idx:=1;
MessageHandler.MessageLine[idx].Visible:=FALSE;
MessageHandler.MessageLine[idx].Editable:=TRUE;
MessageHandler.MessageLine[idx].Text:='Specialmode_1';				(*Ablauf Pallettierer*)
MessageHandler.MessageLine[idx].MsgInt:=1;
MessageHandler.MessageLine[idx].MsgBool:=FALSE;
MessageHandler.MessageLine[idx].MsgTypeEnum:=MsgDataTypeBool;

idx:=idx+1;
MessageHandler.MessageLine[idx].Visible:=FALSE;
MessageHandler.MessageLine[idx].Editable:=TRUE;
MessageHandler.MessageLine[idx].Text:='Specialmode_2';				(*Not used*)
MessageHandler.MessageLine[idx].MsgInt:=2;
MessageHandler.MessageLine[idx].MsgBool:=FALSE;
MessageHandler.MessageLine[idx].MsgTypeEnum:=MsgDataTypeBool;

idx:=idx+1;
MessageHandler.MessageLine[idx].Visible:=FALSE;
MessageHandler.MessageLine[idx].Editable:=TRUE;
MessageHandler.MessageLine[idx].Text:='Specialmode_3';				(*Not used*)
MessageHandler.MessageLine[idx].MsgInt:=3;
MessageHandler.MessageLine[idx].MsgBool:=FALSE;
MessageHandler.MessageLine[idx].MsgTypeEnum:=MsgDataTypeBool;

idx:=idx+1;
MessageHandler.MessageLine[idx].Visible:=FALSE;
MessageHandler.MessageLine[idx].Editable:=TRUE;
MessageHandler.MessageLine[idx].Text:='Specialmode_4';				(*Not used*)
MessageHandler.MessageLine[idx].MsgInt:=4;
MessageHandler.MessageLine[idx].MsgBool:=FALSE;
MessageHandler.MessageLine[idx].MsgTypeEnum:=MsgDataTypeBool;

idx:=idx+1;
MessageHandler.MessageLine[idx].Visible:=FALSE;
MessageHandler.MessageLine[idx].Editable:=TRUE;
MessageHandler.MessageLine[idx].Text:='Specialmode_5';				(*Blister Abstapeln*)
MessageHandler.MessageLine[idx].MsgInt:=5;
MessageHandler.MessageLine[idx].MsgBool:=FALSE;
MessageHandler.MessageLine[idx].MsgTypeEnum:=MsgDataTypeBool;

idx:=idx+1;
MessageHandler.MessageLine[idx].Visible:=gTypeCode=312 OR gTypeCode=499 OR gTypeCode=322;	(*93pol*)(*102pol*)(*160pol*);
MessageHandler.MessageLine[idx].Editable:=TRUE;
MessageHandler.MessageLine[idx].Text:='Specialmode_6';				(*Dummytest*)
MessageHandler.MessageLine[idx].MsgInt:=6;
MessageHandler.MessageLine[idx].MsgBool:=FALSE;
MessageHandler.MessageLine[idx].MsgTypeEnum:=MsgDataTypeBool;

idx:=idx+1;
MessageHandler.MessageLine[idx].Visible:=FALSE;
MessageHandler.MessageLine[idx].Editable:=TRUE;
MessageHandler.MessageLine[idx].Text:='Specialmode_7';				(*Not used*)
MessageHandler.MessageLine[idx].MsgInt:=7;
MessageHandler.MessageLine[idx].MsgBool:=FALSE;
MessageHandler.MessageLine[idx].MsgTypeEnum:=MsgDataTypeBool;

idx:=idx+1;
MessageHandler.MessageLine[idx].Visible:=FALSE;
MessageHandler.MessageLine[idx].Editable:=TRUE;
MessageHandler.MessageLine[idx].Text:='Specialmode_8';				(*Not used*)
MessageHandler.MessageLine[idx].MsgInt:=8;
MessageHandler.MessageLine[idx].MsgBool:=FALSE;
MessageHandler.MessageLine[idx].MsgTypeEnum:=MsgDataTypeBool;

IF 	ModeNo>=1 AND
	ModeNo<=8 THEN
	MessageHandler.MessageLine[ModeNo].MsgBool:=TRUE;
END_IF
END_ACTION

ACTION Msg_SpecialMenu_action:
MessageHandler.Msg.ID:='PM61';
MessageHandler.Msg.Name:='Teil-Abläufe';
MessageHandler.Msg.Text:='Teilablauf auswählen und mit OK starten';
MessageHandler.Msg.Color:=Color.yellow;
MessageHandler.Msg.Station:=0;


MessageHandler(
	Prio:=2, 					(*1=highest, .. , 4=lowest*)
	Btn1Addr:=ADR(MsgOk),		(*Address of Button1 , if Zero then Button is unvisible*)
	Btn2Addr:=ADR(MsgCancel),	(*Address of Button2 , if Zero then Button is unvisible*)
	sVisu:=Visu.Message);

MessageHandler.DisableMultiSelect(sVisu:=Visu.Message);

FOR idx:=1 TO 10 DO
	IF 	MessageHandler.MessageLine[idx].MsgBool THEN
		ModeNo:=idx;
	END_IF
END_FOR
END_ACTION

ACTION Msg_SpecialMenu_exit:
MsgOk:=FALSE;
MsgCancel:=FALSE;
END_ACTION

ACTION SpecialMode01__action:
IF SpecialMode01.State=STATE_WAIT
THEN
	SpecialMode01(Start:=TRUE);

	SFCRun:=TRUE;
(*ELSE*)
END_IF
END_ACTION

ACTION SpecialMode01__exit:
SpecialMode01.Start:=FALSE;
SFCRun:=FALSE;
END_ACTION

ACTION SpecialMode02__action:
IF SpecialMode02.State=STATE_WAIT
THEN
	SpecialMode02(Start:=TRUE);

	SFCRun:=TRUE;
(*ELSE*)
END_IF
END_ACTION

ACTION SpecialMode02__exit:
SpecialMode02.Start:=FALSE;
SFCRun:=FALSE;
END_ACTION

ACTION SpecialMode03__action:
IF SpecialMode03.State=STATE_WAIT
THEN
	SpecialMode03(Start:=TRUE);

	SFCRun:=TRUE;
(*ELSE*)
END_IF
END_ACTION

ACTION SpecialMode03__exit:
SpecialMode03.Start:=FALSE;
SFCRun:=FALSE;
END_ACTION

ACTION SpecialMode04__action:
IF SpecialMode04.State=STATE_WAIT
THEN
	SpecialMode04(Start:=TRUE);

	SFCRun:=TRUE;
(*ELSE*)
END_IF
END_ACTION

ACTION SpecialMode04__exit:
SpecialMode04.Start:=FALSE;
SFCRun:=FALSE;
END_ACTION

ACTION SpecialMode05__action:
IF SpecialMode05.State=STATE_WAIT
THEN
	SpecialMode05(Start:=TRUE);

	SFCRun:=TRUE;
(*ELSE*)
END_IF
END_ACTION

ACTION SpecialMode05__exit:
SpecialMode05.Start:=FALSE;
SFCRun:=FALSE;
END_ACTION

ACTION SpecialMode06__action:
IF SpecialMode06.State=STATE_WAIT
THEN
	SpecialMode06(Start:=TRUE);

	IF	gTypeCode=312 OR		(*93pol*)
		gTypeCode=499 THEN		(*102pol*)
		MP.ST02.DummyPruefung_93pol  := TRUE;
	ELSIF
		gTypeCode=322	THEN	(*160pol*)
		DummyTest_160pol := TRUE;
	END_IF
	SFCRun:=TRUE;
END_IF
END_ACTION

ACTION SpecialMode06__exit:
SpecialMode06.Start:=FALSE;
SFCRun:=FALSE;
DummyTest_160pol := FALSE;
MP.ST02.DummyPruefung_93pol  := FALSE;
END_ACTION

ACTION SpecialMode07__action:
IF SpecialMode07.State=STATE_WAIT
THEN
	SpecialMode07(Start:=TRUE);

	SFCRun:=TRUE;
(*ELSE*)
END_IF
END_ACTION

ACTION SpecialMode07__exit:
SpecialMode07.Start:=FALSE;
SFCRun:=FALSE;
END_ACTION

ACTION SpecialMode08__action:
IF SpecialMode08.State=STATE_WAIT
THEN
	SpecialMode08(Start:=TRUE);

	SFCRun:=TRUE;
(*ELSE*)
END_IF
END_ACTION

ACTION SpecialMode08__exit:
SpecialMode08.Start:=FALSE;
SFCRun:=FALSE;
END_ACTION

ACTION SeqEnd_action:
SFCTime:=TIME_TO_DINT(TIME()-SFCTimeStart);
State:=STATE_OK;
END_ACTION

TRANSITION ModeNo=1:
ModeNo=1
END_TRANSITION

TRANSITION StateOk:
		SFCRun=TRUE
AND SpecialMode01.State=STATE_OK
END_TRANSITION

TRANSITION ModeNo=2:
ModeNo=2
END_TRANSITION

TRANSITION StateOk:
		SFCRun=TRUE
AND SpecialMode02.State=STATE_OK
END_TRANSITION

TRANSITION ModeNo=3:
ModeNo=3
END_TRANSITION

TRANSITION StateOk:
		SFCRun=TRUE
AND SpecialMode03.State=STATE_OK
END_TRANSITION

TRANSITION ModeNo=4:
ModeNo=4
END_TRANSITION

TRANSITION StateOk:
		SFCRun=TRUE
AND SpecialMode04.State=STATE_OK
END_TRANSITION

TRANSITION ModeNo=5:
ModeNo=5
END_TRANSITION

TRANSITION StateOk:
		SFCRun=TRUE
AND SpecialMode05.State=STATE_OK
END_TRANSITION

TRANSITION ModeNo=6:
ModeNo=6
END_TRANSITION

TRANSITION StateOk:
		SFCRun=TRUE
AND SpecialMode06.State=STATE_OK
END_TRANSITION

TRANSITION ModeNo=7:
ModeNo=7
END_TRANSITION

TRANSITION StateOk:
		SFCRun=TRUE
AND SpecialMode07.State=STATE_OK
END_TRANSITION

TRANSITION ModeNo=8:
ModeNo=8
END_TRANSITION

TRANSITION StateOk:
		SFCRun=TRUE
AND SpecialMode08.State=STATE_OK
END_TRANSITION
END_PROGRAM

(* POU Stations/ST_00/ST00_SFCs/_SpecialModeSFCs/SpecialMode02, SFC *)
PROGRAM SpecialMode02 (*Used for: Prozess Kamera *)
(* Date:     Author:   *)

VAR_OUTPUT
	SFCCurrentPOU		: STRING:='SpecialMode02';
	SFCCurrentStep	: STRING:='';
	SFCTime					:	DINT;
  State   				:	DINT;
  Result  				:	DINT;
END_VAR
VAR_INPUT
	Start						:	BOOL;
END_VAR
VAR
	MsgOK				:	BOOL;
	MsgCancel		:	BOOL;
	SFCRun					:	BOOL;
	SFCTimeStart		:	TIME;

	(* Userdefinded area *)


END_VAR
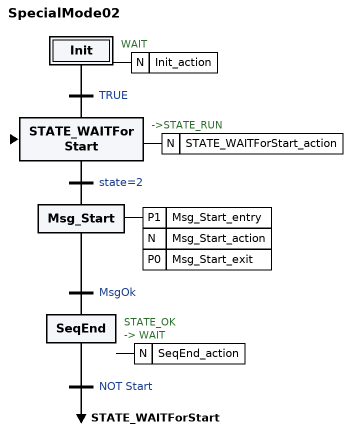
INITIAL_STEP Init: (* WAIT *)
	Init_action(N);
END_STEP
TRANSITION FROM Init TO STATE_WAITForStart := TRUE;
END_TRANSITION
STEP STATE_WAITForStart: (* ->STATE_RUN *)
	STATE_WAITForStart_action(N);
END_STEP
TRANSITION FROM STATE_WAITForStart TO Msg_Start := state=2;
END_TRANSITION
STEP Msg_Start:
	Msg_Start_entry(P1);
	Msg_Start_action(N);
	Msg_Start_exit(P0);
END_STEP
TRANSITION FROM Msg_Start TO SeqEnd := MsgOk;
END_TRANSITION
STEP SeqEnd: (* STATE_OK / -> WAIT *)
	SeqEnd_action(N);
END_STEP
TRANSITION FROM SeqEnd TO STATE_WAITForStart := NOT Start;
END_TRANSITION

ACTION Init_action:
Start:=FALSE;
State:=STATE_WAIT;
END_ACTION

ACTION STATE_WAITForStart_action:
IF Start=TRUE
THEN
	State:=STATE_RUN;
	Result:=RESULT_NON;
	SFCTimeStart:=TIME();
(*ELSE*)
END_IF
END_ACTION

ACTION Msg_Start_entry:
MessageHandler.ClearMessageLines(sVisu:=Visu.Message);
END_ACTION

ACTION Msg_Start_action:
MessageHandler.Msg.ID:='PM51';
MessageHandler.Msg.Name:='SpecialMode02_Start';
MessageHandler.Msg.Text:='Special Mode 2';
MessageHandler.Msg.Color:=Color.yellow;
MessageHandler.Msg.Station:=1;


MessageHandler(
	Prio:=2, 									(*1=highest, .. , 4=lowest*)
	Btn1Addr:=ADR(MsgOk),			(*Address of Button1 , if Zero then Button is unvisible*)
	Btn2Addr:=ADR(MsgCancel),	(*Address of Button2 , if Zero then Button is unvisible*)
	sVisu:=Visu.Message);


MessageHandler.MessageLine[1].Visible:=TRUE;
MessageHandler.MessageLine[1].Editable:=TRUE;
MessageHandler.MessageLine[1].Text:='Kamera Programm ';
MessageHandler.MessageLine[1].MsgTypeEnum:=MsgDataTypeDint;
END_ACTION

ACTION Msg_Start_exit:
MsgOk:=FALSE;
MsgCancel:=FALSE;
SpecialModeProgNu:=MessageHandler.MessageLine[1].MsgInt;
END_ACTION

ACTION SeqEnd_action:
IF 	State=STATE_RUN THEN
	SFCTime:=TIME_TO_DINT(TIME()-SFCTimeStart);
	State:=STATE_OK;
END_IF

IF 	NOT Start THEN
	State:=STATE_WAIT;
END_IF
END_ACTION
END_PROGRAM

(* POU Stations/ST_00/ST00_SFCs/_SpecialModeSFCs/SpecialMode04, SFC *)
PROGRAM SpecialMode04 (*not used*)
(* Date:     Author:   *)

VAR_OUTPUT
	SFCCurrentPOU		: STRING:='SpecialMode04';
	SFCCurrentStep		: STRING:='';
	SFCTime				: DINT;
	State   			: DINT;
	Result  			: DINT;
END_VAR
VAR_INPUT
	Start				: BOOL;
END_VAR
VAR
	MsgOK				: BOOL;
	MsgCancel			: BOOL;
	SFCRun				: BOOL;
	SFCTimeStart		: TIME;
	ResultString		: STRING;
	(* Userdefinded area *)



END_VAR
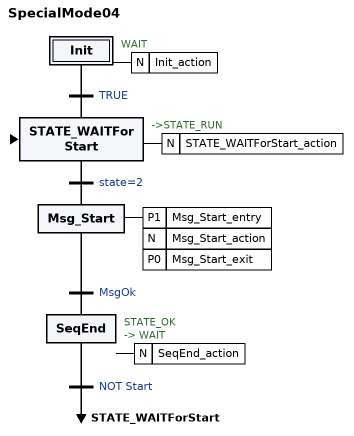
INITIAL_STEP Init: (* WAIT *)
	Init_action(N);
END_STEP
TRANSITION FROM Init TO STATE_WAITForStart := TRUE;
END_TRANSITION
STEP STATE_WAITForStart: (* ->STATE_RUN *)
	STATE_WAITForStart_action(N);
END_STEP
TRANSITION FROM STATE_WAITForStart TO Msg_Start := state=2;
END_TRANSITION
STEP Msg_Start:
	Msg_Start_entry(P1);
	Msg_Start_action(N);
	Msg_Start_exit(P0);
END_STEP
TRANSITION FROM Msg_Start TO SeqEnd := MsgOk;
END_TRANSITION
STEP SeqEnd: (* STATE_OK / -> WAIT *)
	SeqEnd_action(N);
END_STEP
TRANSITION FROM SeqEnd TO STATE_WAITForStart := NOT Start;
END_TRANSITION

ACTION Init_action:
Start:=FALSE;
State:=STATE_WAIT;
END_ACTION

ACTION STATE_WAITForStart_action:
IF Start=TRUE
THEN
	State:=STATE_RUN;
	Result:=RESULT_NON;
	SFCTimeStart:=TIME();
(*ELSE*)
END_IF
END_ACTION

ACTION Msg_Start_entry:
MessageHandler.ClearMessageLines(sVisu:=Visu.Message);
END_ACTION

ACTION Msg_Start_action:
MessageHandler.Msg.ID:='PM52';
MessageHandler.Msg.Name:='SpecialMode04_Start';
MessageHandler.Msg.Text:='Special Mode 4';
MessageHandler.Msg.Color:=Color.yellow;
MessageHandler.Msg.Station:=1;


MessageHandler(
	Prio:=2, 									(*1=highest, .. , 4=lowest*)
	Btn1Addr:=ADR(MsgOk),			(*Address of Button1 , if Zero then Button is unvisible*)
	Btn2Addr:=ADR(MsgCancel),	(*Address of Button2 , if Zero then Button is unvisible*)
	sVisu:=Visu.Message);


MessageHandler.MessageLine[1].Visible:=TRUE;
MessageHandler.MessageLine[1].Editable:=TRUE;
MessageHandler.MessageLine[1].Text:='Kamera Programm ';
MessageHandler.MessageLine[1].MsgTypeEnum:=MsgDataTypeDint;
END_ACTION

ACTION Msg_Start_exit:
MsgOk:=FALSE;
MsgCancel:=FALSE;

SpecialModeProgNu:=MessageHandler.MessageLine[1].MsgInt;
END_ACTION

ACTION SeqEnd_action:
IF 	State=STATE_RUN THEN
	SFCTime:=TIME_TO_DINT(TIME()-SFCTimeStart);
	State:=STATE_OK;
END_IF

IF 	NOT Start THEN
	State:=STATE_WAIT;
END_IF
END_ACTION
END_PROGRAM

(* POU Stations/ST_00/ST00_SFCs/_SpecialModeSFCs/SpecialMode05, SFC *)
PROGRAM SpecialMode05 (*Used for: xxxx *)
(* Date:     Author:   *)

VAR_OUTPUT
	SFCCurrentPOU		: STRING:='SpecialMode05';
	SFCCurrentStep	: STRING:='';
	SFCTime					:	DINT;
  State   				:	DINT;
  Result  				:	DINT;

	ConveyorOn				: BOOL;

END_VAR
VAR_INPUT
	Start						:	BOOL;
END_VAR
VAR
	MsgOK				:	BOOL;
	MsgCancel		:	BOOL;
	SFCRun					:	BOOL;
	SFCTimeStart		:	TIME;

	(* Userdefinded area *)

END_VAR
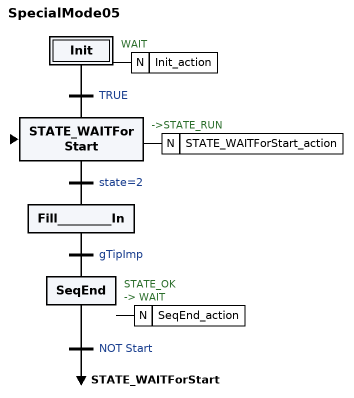
INITIAL_STEP Init: (* WAIT *)
	Init_action(N);
END_STEP
TRANSITION FROM Init TO STATE_WAITForStart := TRUE;
END_TRANSITION
STEP STATE_WAITForStart: (* ->STATE_RUN *)
	STATE_WAITForStart_action(N);
END_STEP
TRANSITION FROM STATE_WAITForStart TO Fill_________In := state=2;
END_TRANSITION
STEP Fill_________In:
END_STEP
TRANSITION FROM Fill_________In TO SeqEnd := gTipImp;
END_TRANSITION
STEP SeqEnd: (* STATE_OK / -> WAIT *)
	SeqEnd_action(N);
END_STEP
TRANSITION FROM SeqEnd TO STATE_WAITForStart := NOT Start;
END_TRANSITION

ACTION Init_action:
Start:=FALSE;
State:=STATE_WAIT;
END_ACTION

ACTION STATE_WAITForStart_action:
IF Start=TRUE
THEN
	State:=STATE_RUN;
	Result:=RESULT_NON;
	SFCTimeStart:=TIME();
(*ELSE*)
END_IF
END_ACTION

ACTION SeqEnd_action:
IF 	State=STATE_RUN THEN
	SFCTime:=TIME_TO_DINT(TIME()-SFCTimeStart);
	State:=STATE_OK;
END_IF

IF 	NOT Start THEN
	State:=STATE_WAIT;
END_IF
END_ACTION
END_PROGRAM

(* POU Stations/ST_00/ST00_SFCs/_SpecialModeSFCs/SpecialMode07, SFC *)
PROGRAM SpecialMode07 (*Used for: xxxx *)
(* Date:     Author:   *)

VAR_OUTPUT
	SFCCurrentPOU		: STRING:='SpecialMode07';
	SFCCurrentStep	: STRING:='';
	SFCTime					:	DINT;
  State   				:	DINT;
  Result  				:	DINT;
END_VAR
VAR_INPUT
	Start						:	BOOL;
END_VAR
VAR
	MsgOK				:	BOOL;
	MsgCancel		:	BOOL;
	SFCRun					:	BOOL;
	SFCTimeStart		:	TIME;
  Delay         :TON;

	(* Userdefinded area *)


END_VAR
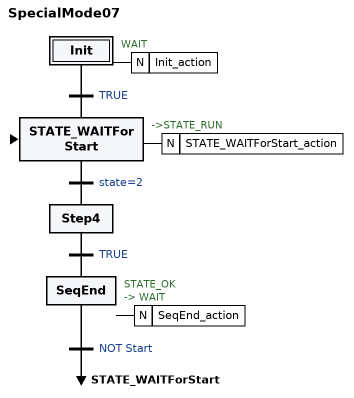
INITIAL_STEP Init: (* WAIT *)
	Init_action(N);
END_STEP
TRANSITION FROM Init TO STATE_WAITForStart := TRUE;
END_TRANSITION
STEP STATE_WAITForStart: (* ->STATE_RUN *)
	STATE_WAITForStart_action(N);
END_STEP
TRANSITION FROM STATE_WAITForStart TO Step4 := state=2;
END_TRANSITION
STEP Step4:
END_STEP
TRANSITION FROM Step4 TO SeqEnd := TRUE;
END_TRANSITION
STEP SeqEnd: (* STATE_OK / -> WAIT *)
	SeqEnd_action(N);
END_STEP
TRANSITION FROM SeqEnd TO STATE_WAITForStart := NOT Start;
END_TRANSITION

ACTION Init_action:
Start:=FALSE;
State:=STATE_WAIT;
END_ACTION

ACTION STATE_WAITForStart_action:
IF Start=TRUE
THEN
	State:=STATE_RUN;
	Result:=RESULT_NON;
	SFCTimeStart:=TIME();
(*ELSE*)
END_IF
END_ACTION

ACTION SeqEnd_action:
IF 	State=STATE_RUN THEN
	SFCTime:=TIME_TO_DINT(TIME()-SFCTimeStart);
	State:=STATE_OK;
END_IF

IF 	NOT Start THEN
	State:=STATE_WAIT;
END_IF
END_ACTION
END_PROGRAM

(* POU Stations/ST_00/ST00_SFCs/_SpecialModeSFCs/SpecialMode08, SFC *)
PROGRAM SpecialMode08 (*Used for: xxxx *)
(* Date:     Author:   *)

VAR_OUTPUT
	SFCCurrentPOU		: STRING:='SpecialMode08';
	SFCCurrentStep	: STRING:='';
	SFCTime					:	DINT;
  State   				:	DINT;
  Result  				:	DINT;
END_VAR
VAR_INPUT
	Start						:	BOOL;
END_VAR
VAR
	MsgOK				:	BOOL;
	MsgCancel		:	BOOL;
	SFCRun					:	BOOL;
	SFCTimeStart		:	TIME;

	(* Userdefinded area *)
	TestDint1:DINT:=12;
	TestDint2:DINT:=34;
	IntPosIdx:	DINT;

END_VAR
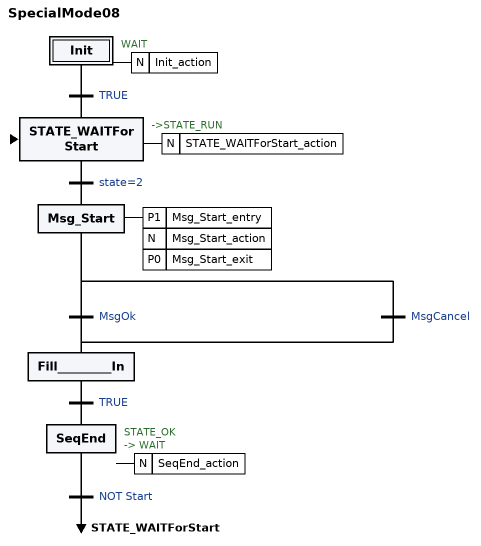
INITIAL_STEP Init: (* WAIT *)
	Init_action(N);
END_STEP
TRANSITION FROM Init TO STATE_WAITForStart := TRUE;
END_TRANSITION
STEP STATE_WAITForStart: (* ->STATE_RUN *)
	STATE_WAITForStart_action(N);
END_STEP
TRANSITION FROM STATE_WAITForStart TO Msg_Start := state=2;
END_TRANSITION
STEP Msg_Start:
	Msg_Start_entry(P1);
	Msg_Start_action(N);
	Msg_Start_exit(P0);
END_STEP
TRANSITION FROM Msg_Start TO Fill_________In := MsgOk;
END_TRANSITION
TRANSITION FROM Msg_Start TO Fill_________In := MsgCancel;
END_TRANSITION
STEP Fill_________In:
END_STEP
TRANSITION FROM Fill_________In TO SeqEnd := TRUE;
END_TRANSITION
STEP SeqEnd: (* STATE_OK / -> WAIT *)
	SeqEnd_action(N);
END_STEP
TRANSITION FROM SeqEnd TO STATE_WAITForStart := NOT Start;
END_TRANSITION

ACTION Init_action:
Start:=FALSE;
State:=STATE_WAIT;
END_ACTION

ACTION STATE_WAITForStart_action:
IF Start=TRUE
THEN
	State:=STATE_RUN;
	Result:=RESULT_NON;
	SFCTimeStart:=TIME();
(*ELSE*)
END_IF
END_ACTION

ACTION Msg_Start_entry:
MessageHandler.ClearMessageLines(sVisu:=Visu.Message);
IntPosIdx:=1;
END_ACTION

ACTION Msg_Start_action:
MessageHandler.Msg.ID:='PM53';
MessageHandler.Msg.Name:='SpecialMode08_Start';
MessageHandler.Msg.Text:='Teilautomatik Ablauf08: Test Messagehandler';
MessageHandler.Msg.Color:=Color.yellow;
MessageHandler.Msg.Station:=1;


MessageHandler(
	Prio:=2, 									(*1=highest, .. , 4=lowest*)
	Btn1Addr:=ADR(MsgOk),			(*Address of Button1 , if Zero then Button is unvisible*)
	Btn2Addr:=ADR(MsgCancel),	(*Address of Button2 , if Zero then Button is unvisible*)
	sVisu:=Visu.Message);


MessageHandler.MessageLine[1].Visible:=TRUE;
MessageHandler.MessageLine[1].Editable:=TRUE;
MessageHandler.MessageLine[1].Text:='TestZeile1';
MessageHandler.MessageLine[1].MsgInt:=TestDint1;
MessageHandler.MessageLine[1].MsgTypeEnum:=MsgDataTypeDint;

MessageHandler.MessageLine[2].Visible:=TRUE;
MessageHandler.MessageLine[2].Editable:=TRUE;
MessageHandler.MessageLine[2].Text:='TestZeile2';
MessageHandler.MessageLine[2].MsgInt:=TestDint2;
MessageHandler.MessageLine[2].MsgTypeEnum:=MsgDataTypeDint;
END_ACTION

ACTION Msg_Start_exit:
MsgOk:=FALSE;
MsgCancel:=FALSE;

TestDint1:=MessageHandler.MessageLine[1].MsgInt;
TestDint2:=MessageHandler.MessageLine[2].MsgInt;
END_ACTION

ACTION SeqEnd_action:
IF 	State=STATE_RUN THEN
	SFCTime:=TIME_TO_DINT(TIME()-SFCTimeStart);
	State:=STATE_OK;
END_IF


IF 	NOT Start THEN
	State:=STATE_WAIT;
END_IF
END_ACTION
END_PROGRAM

(* POU Stations/ST_00/ST00_SFCs/HomePositionSFC, SFC *)
PROGRAM HomePositionSFC


VAR_OUTPUT
	SFCCurrentPOU		: STRING:='HomePositionSFC';
	SFCCurrentStep		: STRING:='';
	SFCTime				: DINT;
	State   			: StateObject	:= STATE_WAIT;
	Result  			: StateResult;
END_VAR
VAR_INPUT
	Start				: BOOL;
END_VAR
VAR
	MsgOK				: BOOL;
	MsgCancel			: BOOL;
	SFCRun				: BOOL;
	SFCTimeStart		: TIME;
	Error				: ErrorStruct;
	(* Userdefinded area *)
	SFCRun01			: BOOL;
	SFCRun02			: BOOL;
	SFCRun03			: BOOL;
	SFCRun04			: BOOL;
	SFCRun05			: BOOL;
	SFCRun08			: BOOL;
	idx					: INT;


END_VAR
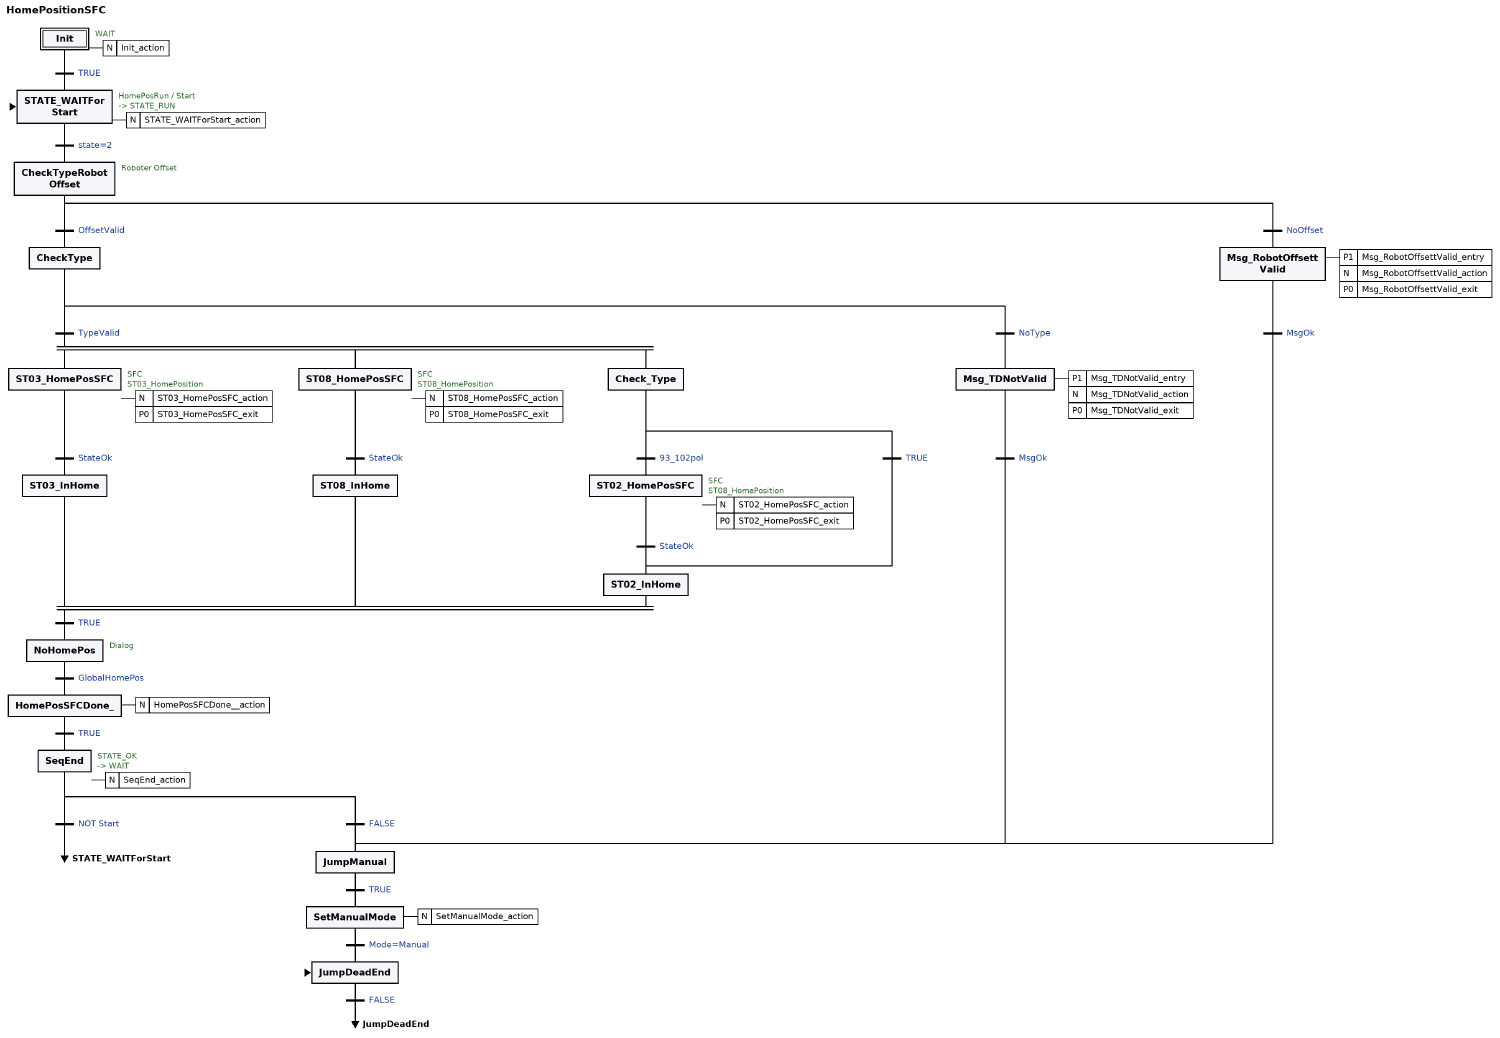
INITIAL_STEP Init: (* WAIT *)
	Init_action(N);
END_STEP
TRANSITION FROM Init TO STATE_WAITForStart := TRUE;
END_TRANSITION
STEP STATE_WAITForStart: (* HomePosRun / Start / -> STATE_RUN *)
	STATE_WAITForStart_action(N);
END_STEP
TRANSITION FROM STATE_WAITForStart TO CheckTypeRobotOffset := state=2;
END_TRANSITION
STEP CheckTypeRobotOffset: (* Roboter Offset *)
END_STEP
TRANSITION FROM CheckTypeRobotOffset TO CheckType := OffsetValid;
END_TRANSITION
TRANSITION FROM CheckTypeRobotOffset TO Msg_RobotOffsettValid := NoOffset;
END_TRANSITION
STEP CheckType:
END_STEP
TRANSITION FROM CheckType TO (ST03_HomePosSFC, ST08_HomePosSFC, Check_Type) := TypeValid;
END_TRANSITION
TRANSITION FROM CheckType TO Msg_TDNotValid := NoType;
END_TRANSITION
STEP Msg_TDNotValid:
	Msg_TDNotValid_entry(P1);
	Msg_TDNotValid_action(N);
	Msg_TDNotValid_exit(P0);
END_STEP
TRANSITION FROM Msg_TDNotValid TO JumpManual := MsgOk;
END_TRANSITION
STEP Msg_RobotOffsettValid:
	Msg_RobotOffsettValid_entry(P1);
	Msg_RobotOffsettValid_action(N);
	Msg_RobotOffsettValid_exit(P0);
END_STEP
TRANSITION FROM Msg_RobotOffsettValid TO JumpManual := MsgOk;
END_TRANSITION
STEP ST03_HomePosSFC: (* SFC / ST03_HomePosition *)
	ST03_HomePosSFC_action(N);
	ST03_HomePosSFC_exit(P0);
END_STEP
TRANSITION FROM ST03_HomePosSFC TO ST03_InHome := StateOk;
END_TRANSITION
STEP ST03_InHome:
END_STEP
STEP ST08_HomePosSFC: (* SFC / ST08_HomePosition *)
	ST08_HomePosSFC_action(N);
	ST08_HomePosSFC_exit(P0);
END_STEP
TRANSITION FROM ST08_HomePosSFC TO ST08_InHome := StateOk;
END_TRANSITION
STEP ST08_InHome:
END_STEP
STEP Check_Type:
END_STEP
TRANSITION FROM Check_Type TO ST02_HomePosSFC := 93_102pol;
END_TRANSITION
TRANSITION FROM Check_Type TO ST02_InHome := TRUE;
END_TRANSITION
STEP ST02_HomePosSFC: (* SFC / ST08_HomePosition *)
	ST02_HomePosSFC_action(N);
	ST02_HomePosSFC_exit(P0);
END_STEP
TRANSITION FROM ST02_HomePosSFC TO ST02_InHome := StateOk;
END_TRANSITION
STEP ST02_InHome:
END_STEP
TRANSITION FROM (ST03_InHome, ST08_InHome, ST02_InHome) TO NoHomePos := TRUE;
END_TRANSITION
STEP NoHomePos: (* Dialog *)
END_STEP
TRANSITION FROM NoHomePos TO HomePosSFCDone_ := GlobalHomePos;
END_TRANSITION
STEP HomePosSFCDone_:
	HomePosSFCDone__action(N);
END_STEP
TRANSITION FROM HomePosSFCDone_ TO SeqEnd := TRUE;
END_TRANSITION
STEP SeqEnd: (* STATE_OK / -> WAIT *)
	SeqEnd_action(N);
END_STEP
TRANSITION FROM SeqEnd TO STATE_WAITForStart := NOT Start;
END_TRANSITION
TRANSITION FROM SeqEnd TO JumpManual := FALSE;
END_TRANSITION
STEP JumpManual:
END_STEP
TRANSITION FROM JumpManual TO SetManualMode := TRUE;
END_TRANSITION
STEP SetManualMode:
	SetManualMode_action(N);
END_STEP
TRANSITION FROM SetManualMode TO JumpDeadEnd := Mode=Manual;
END_TRANSITION
STEP JumpDeadEnd:
END_STEP
TRANSITION FROM JumpDeadEnd TO JumpDeadEnd := FALSE;
END_TRANSITION

ACTION Init_action:
Start:=FALSE;
State:=STATE_WAIT;
END_ACTION

ACTION STATE_WAITForStart_action:
IF	(ModeSelect.Mode=MODE_HOME_POS_RUN OR
	Start) AND
	NOT PLC_PRG.GlobalHomePos THEN
	State:=STATE_RUN;
	Result:=RESULT_NON;
	SFCTimeStart:=TIME();
END_IF

SFCRun		:=FALSE;
SFCRun01	:=FALSE;
SFCRun02	:=FALSE;
SFCRun03	:=FALSE;
SFCRun04	:=FALSE;
SFCRun05	:=FALSE;
END_ACTION

ACTION Msg_TDNotValid_entry:
FOR idx:=1 TO 8
DO
	MessageHandler.MessageLine[idx].Visible:=FALSE;
	MessageHandler.MessageLine[idx].Editable:=FALSE;
	MessageHandler.MessageLine[idx].Text:='';
	MessageHandler.MessageLine[idx].MsgInt:=0;
	MessageHandler.MessageLine[idx].MsgTypeEnum:=MsgDataTypeDint;

END_FOR
END_ACTION

ACTION Msg_TDNotValid_action:
MessageHandler.Msg.ID:='PM10';
MessageHandler.Msg.Name:='TDNotValid';
MessageHandler.Msg.Text:='Typdaten nicht gültig, bitte laden!';
MessageHandler.Msg.Text:= CONCAT(MessageHandler.Msg.Text,'$r --> weiter mit <OK>');
MessageHandler.Msg.Color:=Color.yellow;
MessageHandler.Msg.Station:=0;
MessageHandler.MsgButton1Text:='continue';

MessageHandler(
	Prio:=1, 						(*1=highest, .. , 4=lowest*)
	Btn1Addr:=ADR(MsgOk),		(*Address of Button1 , if Zero then Button is unvisible*)
	Btn2Addr:=0,					(*Address of Button2 , if Zero then Button is unvisible*)
	sVisu:=Visu.Message);
END_ACTION

ACTION Msg_TDNotValid_exit:
MsgOk:=FALSE;
MsgCancel:=FALSE;
END_ACTION

ACTION Msg_RobotOffsettValid_entry:
MessageHandler.ClearMessageLines(sVisu:=Visu.Message);
END_ACTION

ACTION Msg_RobotOffsettValid_action:
MessageHandler.Msg.ID:='PM11';
MessageHandler.Msg.Name:='TDRoffsetbotOValid';
MessageHandler.Msg.Text:='Typdaten Roboter Offset nicht gültig, bitte laden!';
MessageHandler.Msg.Text:= CONCAT(MessageHandler.Msg.Text,'$r --> weiter mit <OK>');

MessageHandler.Msg.Color:=Color.yellow;
MessageHandler.Msg.Station:=0;


MessageHandler(
	Prio:=1, 								(*1=highest, .. , 4=lowest*)
	Btn1Addr:=ADR(MsgOk),		(*Address of Button1 , if Zero then Button is unvisible*)
	Btn2Addr:=0,						(*Address of Button2 , if Zero then Button is unvisible*)
	sVisu:=Visu.Message);
END_ACTION

ACTION Msg_RobotOffsettValid_exit:
MsgOk:=FALSE;
MsgCancel:=FALSE;
END_ACTION

ACTION ST03_HomePosSFC_action:
IF ST03_HomePosition.State=STATE_WAIT
THEN
	ST03_HomePosition(Start:=TRUE);

	SFCRun03:=TRUE;
(*ELSE*)
END_IF
END_ACTION

ACTION ST03_HomePosSFC_exit:
ST03_HomePosition.Start:=FALSE;
SFCRun03:=FALSE;
END_ACTION

ACTION ST08_HomePosSFC_action:
IF ST08_HomePosition.State=STATE_WAIT
THEN
	SFCRun08:=TRUE;
	ST08_HomePosition.Start:=TRUE;


(*ELSE*)
END_IF
END_ACTION

ACTION ST08_HomePosSFC_exit:
ST08_HomePosition.Start:=FALSE;
SFCRun08:=FALSE;
END_ACTION

ACTION ST02_HomePosSFC_action:
IF ST02_HomePosition.State=STATE_WAIT THEN
	ST02_HomePosition.Start:=TRUE;
	SFCRun02:=TRUE;
END_IF
END_ACTION

ACTION ST02_HomePosSFC_exit:
ST02_HomePosition.Start:=FALSE;
SFCRun02:=FALSE;
END_ACTION

ACTION HomePosSFCDone__action:
gHomePosSFCDone:=TRUE;
END_ACTION

ACTION SeqEnd_action:
IF 	NOT Start THEN
	State:=STATE_WAIT;
END_IF
END_ACTION

ACTION SetManualMode_action:
ModeSelect.AskForManual:=TRUE;
END_ACTION

TRANSITION OffsetValid:
   gRobotOffset > 0
(*OR gRobotOffset =1000
OR gRobotOffset =2000
OR gRobotOffset =3000
OR gRobotOffset =4000
OR gRobotOffset =5000
OR gRobotOffset =6000
OR gRobotOffset =7000
OR gRobotOffset =19000
OR gRobotOffset =25000
OR gRobotOffset =26000
OR gRobotOffset =27000
OR gRobotOffset =28000
OR gRobotOffset =29000
OR gRobotOffset =30000
OR gRobotOffset =35000*)
END_TRANSITION

TRANSITION TypeValid:
gTypeDataValid
END_TRANSITION

TRANSITION NoType:
TRUE
END_TRANSITION

TRANSITION NoOffset:
TRUE
END_TRANSITION

TRANSITION StateOk:
		SFCRun03=TRUE
AND ST03_HomePosition.State=STATE_OK
END_TRANSITION

TRANSITION StateOk:
		SFCRun08=TRUE
AND ST08_HomePosition.State=STATE_OK
END_TRANSITION

TRANSITION 93_102pol:
gTypeCode=4991 OR 	(*102pol*)
gTypeCode=312		(*93pol*)
END_TRANSITION

TRANSITION StateOk:
SFCRun02 AND
ST02_HomePosition.State=STATE_OK
END_TRANSITION

TRANSITION GlobalHomePos:
PLC_PRG.GlobalHomePos
END_TRANSITION

TRANSITION Mode=Manual:
ModeSelect.Mode=MODE_MANUAL
END_TRANSITION
END_PROGRAM

(* POU Stations/ST_03_Ruestsaetze/ST_03_SFCs/ST03_HomePosition, SFC *)
PROGRAM ST03_HomePosition

VAR_OUTPUT
	SFCCurrentPOU		: STRING:='ST03_HomePosition';
	SFCCurrentStep		: STRING:='';
	SFCTime				: DINT;
	State   			: StateObject	:= STATE_WAIT;
	Result  			: StateResult;

END_VAR
VAR_INPUT
	Start				: BOOL;
END_VAR
VAR
	MsgOK				: BOOL;
	MsgCancel			: BOOL;
	SFCRun				: BOOL;
	SFCTimeStart		: TIME;
	(* Userdefinded area *)

END_VAR
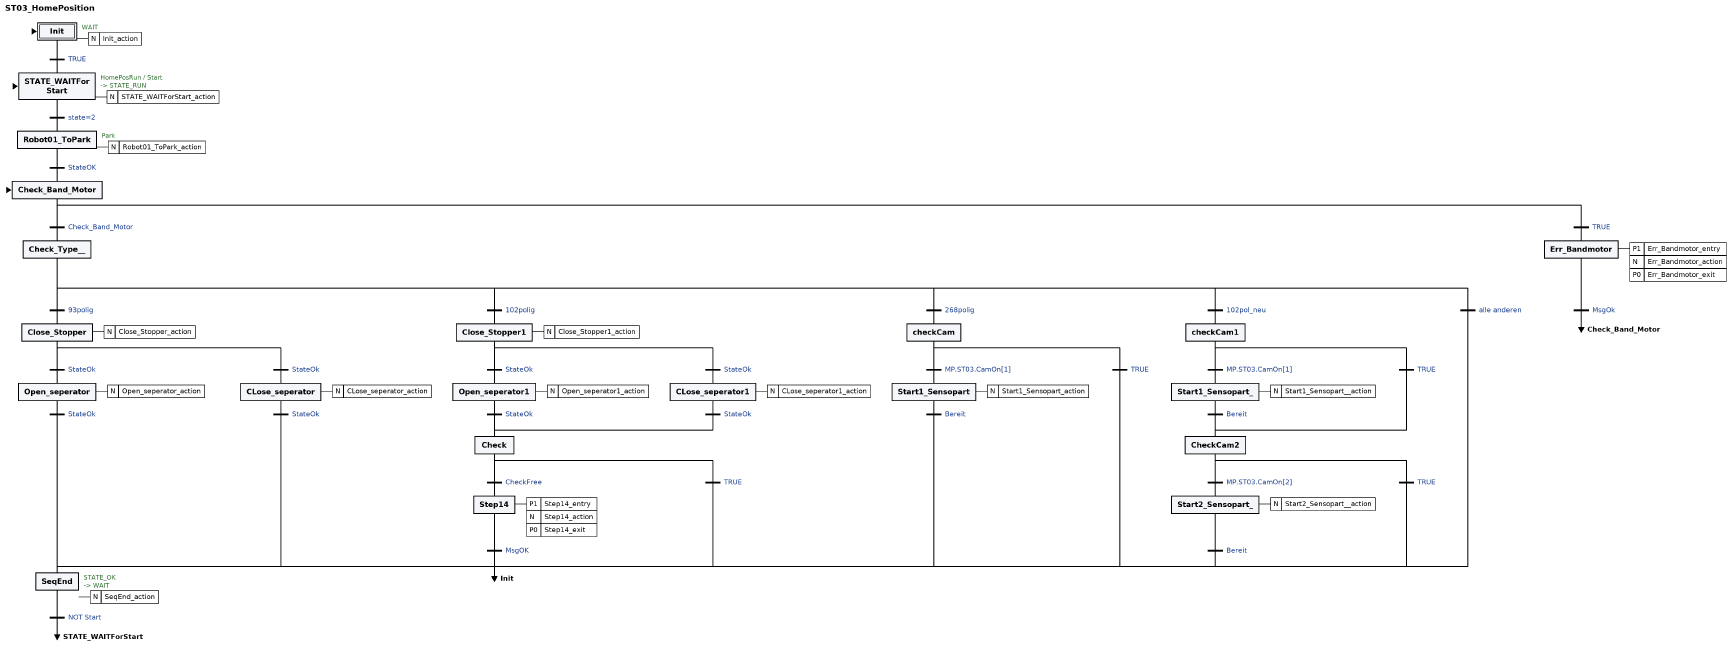
INITIAL_STEP Init: (* WAIT *)
	Init_action(N);
END_STEP
TRANSITION FROM Init TO STATE_WAITForStart := TRUE;
END_TRANSITION
STEP STATE_WAITForStart: (* HomePosRun / Start / -> STATE_RUN *)
	STATE_WAITForStart_action(N);
END_STEP
TRANSITION FROM STATE_WAITForStart TO Robot01_ToPark := state=2;
END_TRANSITION
STEP Robot01_ToPark: (* Park *)
	Robot01_ToPark_action(N);
END_STEP
TRANSITION FROM Robot01_ToPark TO Check_Band_Motor := StateOK;
END_TRANSITION
STEP Check_Band_Motor:
END_STEP
TRANSITION FROM Check_Band_Motor TO Check_Type__ := Check_Band_Motor;
END_TRANSITION
TRANSITION FROM Check_Band_Motor TO Err_Bandmotor := TRUE;
END_TRANSITION
STEP Err_Bandmotor:
	Err_Bandmotor_entry(P1);
	Err_Bandmotor_action(N);
	Err_Bandmotor_exit(P0);
END_STEP
TRANSITION FROM Err_Bandmotor TO Check_Band_Motor := MsgOk;
END_TRANSITION
STEP Check_Type__:
END_STEP
TRANSITION FROM Check_Type__ TO Close_Stopper := 93polig;
END_TRANSITION
TRANSITION FROM Check_Type__ TO Close_Stopper1 := 102polig;
END_TRANSITION
TRANSITION FROM Check_Type__ TO checkCam := 268polig;
END_TRANSITION
TRANSITION FROM Check_Type__ TO checkCam1 := 102pol_neu;
END_TRANSITION
TRANSITION FROM Check_Type__ TO SeqEnd := alle anderen;
END_TRANSITION
STEP Close_Stopper:
	Close_Stopper_action(N);
END_STEP
TRANSITION FROM Close_Stopper TO Open_seperator := StateOk;
END_TRANSITION
TRANSITION FROM Close_Stopper TO CLose_seperator := StateOk;
END_TRANSITION
STEP Open_seperator:
	Open_seperator_action(N);
END_STEP
TRANSITION FROM Open_seperator TO SeqEnd := StateOk;
END_TRANSITION
STEP CLose_seperator:
	CLose_seperator_action(N);
END_STEP
TRANSITION FROM CLose_seperator TO SeqEnd := StateOk;
END_TRANSITION
STEP Close_Stopper1:
	Close_Stopper1_action(N);
END_STEP
TRANSITION FROM Close_Stopper1 TO Open_seperator1 := StateOk;
END_TRANSITION
TRANSITION FROM Close_Stopper1 TO CLose_seperator1 := StateOk;
END_TRANSITION
STEP Open_seperator1:
	Open_seperator1_action(N);
END_STEP
TRANSITION FROM Open_seperator1 TO Check := StateOk;
END_TRANSITION
STEP CLose_seperator1:
	CLose_seperator1_action(N);
END_STEP
TRANSITION FROM CLose_seperator1 TO Check := StateOk;
END_TRANSITION
STEP Check:
END_STEP
TRANSITION FROM Check TO Step14 := CheckFree;
END_TRANSITION
TRANSITION FROM Check TO SeqEnd := TRUE;
END_TRANSITION
STEP Step14:
	Step14_entry(P1);
	Step14_action(N);
	Step14_exit(P0);
END_STEP
TRANSITION FROM Step14 TO Init := MsgOK;
END_TRANSITION
STEP checkCam:
END_STEP
TRANSITION FROM checkCam TO Start1_Sensopart := MP.ST03.CamOn[1];
END_TRANSITION
TRANSITION FROM checkCam TO SeqEnd := TRUE;
END_TRANSITION
STEP Start1_Sensopart:
	Start1_Sensopart_action(N);
END_STEP
TRANSITION FROM Start1_Sensopart TO SeqEnd := Bereit;
END_TRANSITION
STEP checkCam1:
END_STEP
TRANSITION FROM checkCam1 TO Start1_Sensopart_ := MP.ST03.CamOn[1];
END_TRANSITION
TRANSITION FROM checkCam1 TO CheckCam2 := TRUE;
END_TRANSITION
STEP Start1_Sensopart_:
	Start1_Sensopart__action(N);
END_STEP
TRANSITION FROM Start1_Sensopart_ TO CheckCam2 := Bereit;
END_TRANSITION
STEP CheckCam2:
END_STEP
TRANSITION FROM CheckCam2 TO Start2_Sensopart_ := MP.ST03.CamOn[2];
END_TRANSITION
TRANSITION FROM CheckCam2 TO SeqEnd := TRUE;
END_TRANSITION
STEP Start2_Sensopart_:
	Start2_Sensopart__action(N);
END_STEP
TRANSITION FROM Start2_Sensopart_ TO SeqEnd := Bereit;
END_TRANSITION
STEP SeqEnd: (* STATE_OK / -> WAIT *)
	SeqEnd_action(N);
END_STEP
TRANSITION FROM SeqEnd TO STATE_WAITForStart := NOT Start;
END_TRANSITION

ACTION Init_action:
Start:=FALSE;
State:=STATE_WAIT;
END_ACTION

ACTION STATE_WAITForStart_action:
IF	( Start = TRUE )
THEN
	State:=STATE_RUN;
	Result:=RESULT_NON;
	SFCTimeStart:=TIME();
ELSE
	;
END_IF
END_ACTION

ACTION Robot01_ToPark_action:
Robot01.PosNo:=POS_PARK;
Robot01.PosOffset:=gRobotOffset;
Robot01.Override:=MP.ST00.Override;
Robot01.SetToolOn:=FALSE;
Robot01.SetToolOff:=FALSE;
Robot01.ExecuteMove:=TRUE;
END_ACTION

ACTION Err_Bandmotor_entry:
MessageHandler.ClearMessageLines(sVisu:=Visu.Message);
END_ACTION

ACTION Err_Bandmotor_action:
MessageHandler.Msg.ID:='PM100';
MessageHandler.Msg.Name:='Fehler Bandmotor';
MessageHandler.Msg.Text:='Fehler Bandmotor';
MessageHandler.Msg.Color:=Color.red;
MessageHandler.Msg.Station:=1;


MessageHandler(
	Prio:=2, 							(*1=highest, .. , 4=lowest*)
	Btn1Addr:=ADR(MsgOk),			(*Address of Button1 , if Zero then Button is unvisible*)
	Btn2Addr:=,						(*Address of Button2 , if Zero then Button is unvisible*)
	sVisu:=Visu.Message);
END_ACTION

ACTION Err_Bandmotor_exit:
MsgOk:=FALSE;
MsgCancel:=FALSE;
ST03_51_M1.Reset:=TRUE;
END_ACTION

ACTION Close_Stopper_action:
ST00_74_Y2_4.MoveInit:=TRUE;
END_ACTION

ACTION Open_seperator_action:
ST00_74_Y2_5.MoveInit:=TRUE;
END_ACTION

ACTION CLose_seperator_action:
ST00_74_Y2_5.MoveWork:=TRUE;
END_ACTION

ACTION Close_Stopper1_action:
ST00_74_Y2_4.MoveInit:=TRUE;
END_ACTION

ACTION Open_seperator1_action:
ST00_74_Y2_5.MoveInit:=TRUE;
END_ACTION

ACTION CLose_seperator1_action:
ST00_74_Y2_5.MoveWork:=TRUE;
END_ACTION

ACTION Step14_entry:
MessageHandler.ClearMessageLines(sVisu:=Visu.Message);
END_ACTION

ACTION Step14_action:
MessageHandler.Msg.ID:='PM102';
MessageHandler.Msg.Name:='Vereinzler beide Positionen besetzt';
MessageHandler.Msg.Text:='Vereinzler beide Positionen besetzt';
MessageHandler.Msg.Color:=Color.red;
MessageHandler.Msg.Station:=1;


MessageHandler(
	Prio:=2, 							(*1=highest, .. , 4=lowest*)
	Btn1Addr:=ADR(MsgOk),			(*Address of Button1 , if Zero then Button is unvisible*)
	Btn2Addr:=,						(*Address of Button2 , if Zero then Button is unvisible*)
	sVisu:=Visu.Message);
END_ACTION

ACTION Step14_exit:
MsgOk:=FALSE;
MsgCancel:=FALSE;
END_ACTION

ACTION Start1_Sensopart_action:
ST03_8_100_A1.JobNo := TD.Sensopart_CamProgNo ;
ST03_8_100_A1.st_ctrl_in.b_init := TRUE;
END_ACTION

ACTION Start1_Sensopart__action:
ST03_8_100_A1.JobNo := TD.Sensopart_CamProgNo ;
ST03_8_100_A1.st_ctrl_in.b_init := TRUE;
END_ACTION

ACTION Start2_Sensopart__action:
ST03_8_103_A1.JobNo := TD.Sensopart2_CamProgNo ;
ST03_8_103_A1.st_ctrl_in.b_init := TRUE;
END_ACTION

ACTION SeqEnd_action:
IF 	State=STATE_RUN THEN
	SFCTime:=TIME_TO_DINT(TIME()-SFCTimeStart);
	State:=STATE_OK;
END_IF

IF 	NOT Start THEN
	State:=STATE_WAIT;
END_IF
END_ACTION

TRANSITION StateOK:
Robot01.State=STATE_OK
END_TRANSITION

TRANSITION Check_Band_Motor:
NOT ST03_51_M1.Error_ (*AND
ST03_51_M1.On*)
END_TRANSITION

TRANSITION 93polig:
gTypeCode=312	(*93pol*)
END_TRANSITION

TRANSITION StateOk:
ST00_74_Y2_4.State=STATE_OK AND
NOT ST00_72_X1_3.BitInToCheck
END_TRANSITION

TRANSITION StateOk:
ST00_74_Y2_5.State=STATE_OK
END_TRANSITION

TRANSITION StateOk:
ST00_74_Y2_4.State=STATE_OK
END_TRANSITION

TRANSITION StateOk:
ST00_74_Y2_5.State=STATE_OK
END_TRANSITION

TRANSITION 102polig:
gTypeCode=4991	(*102pol*)
END_TRANSITION

TRANSITION StateOk:
ST00_74_Y2_4.State=STATE_OK AND
NOT ST02_FDB_80_B02.BitInToCheck
END_TRANSITION

TRANSITION StateOk:
ST00_74_Y2_5.State=STATE_OK
END_TRANSITION

TRANSITION StateOk:
ST00_74_Y2_4.State=STATE_OK
END_TRANSITION

TRANSITION StateOk:
ST00_74_Y2_5.State=STATE_OK
END_TRANSITION

TRANSITION CheckFree:
ST02_FDB_80_B02.BitInToCheck AND
ST00_72_X1_3.BitInToCheck
END_TRANSITION

TRANSITION 268polig:
gTypeCode=5841 	(*268pol*)
END_TRANSITION

TRANSITION Bereit:
ST03_8_100_A1.st_ctrl_out.b_bereit (*Kamera Farberkennung Ehternet*)
END_TRANSITION

TRANSITION 102pol_neu:
gTypeCode=4993	(*102pol neu*)
END_TRANSITION

TRANSITION Bereit:
ST03_8_100_A1.st_ctrl_out.b_bereit  (*Kamera Farberkennung Ehternet*)
END_TRANSITION

TRANSITION Bereit:
ST03_8_103_A1.st_ctrl_out.b_bereit  (*Kamera Farberkennung Ehternet*)
END_TRANSITION

TRANSITION alle anderen:
TRUE
END_TRANSITION
END_PROGRAM

(* POU Stations/ST_08_Palettierer/ST_08_SFCs/ST08_HomePosition, SFC *)
PROGRAM ST08_HomePosition


VAR_OUTPUT
	SFCCurrentPOU		: STRING:='ST08_HomePosition';
	SFCCurrentStep		: STRING:='';
	SFCTime				: DINT;
	State   			: StateObject	:= STATE_WAIT;
	Result  			: StateResult;
END_VAR
VAR_INPUT
	Start				: BOOL;
END_VAR
VAR
	MsgOK				: BOOL;
	MsgCancel			: BOOL;
	SFCRun				: BOOL;
	SFCTimeStart		: TIME;
	(* Userdefinded area *)
	MsgString      		:STRING;
	MsgID		      	:STRING(20);
END_VAR
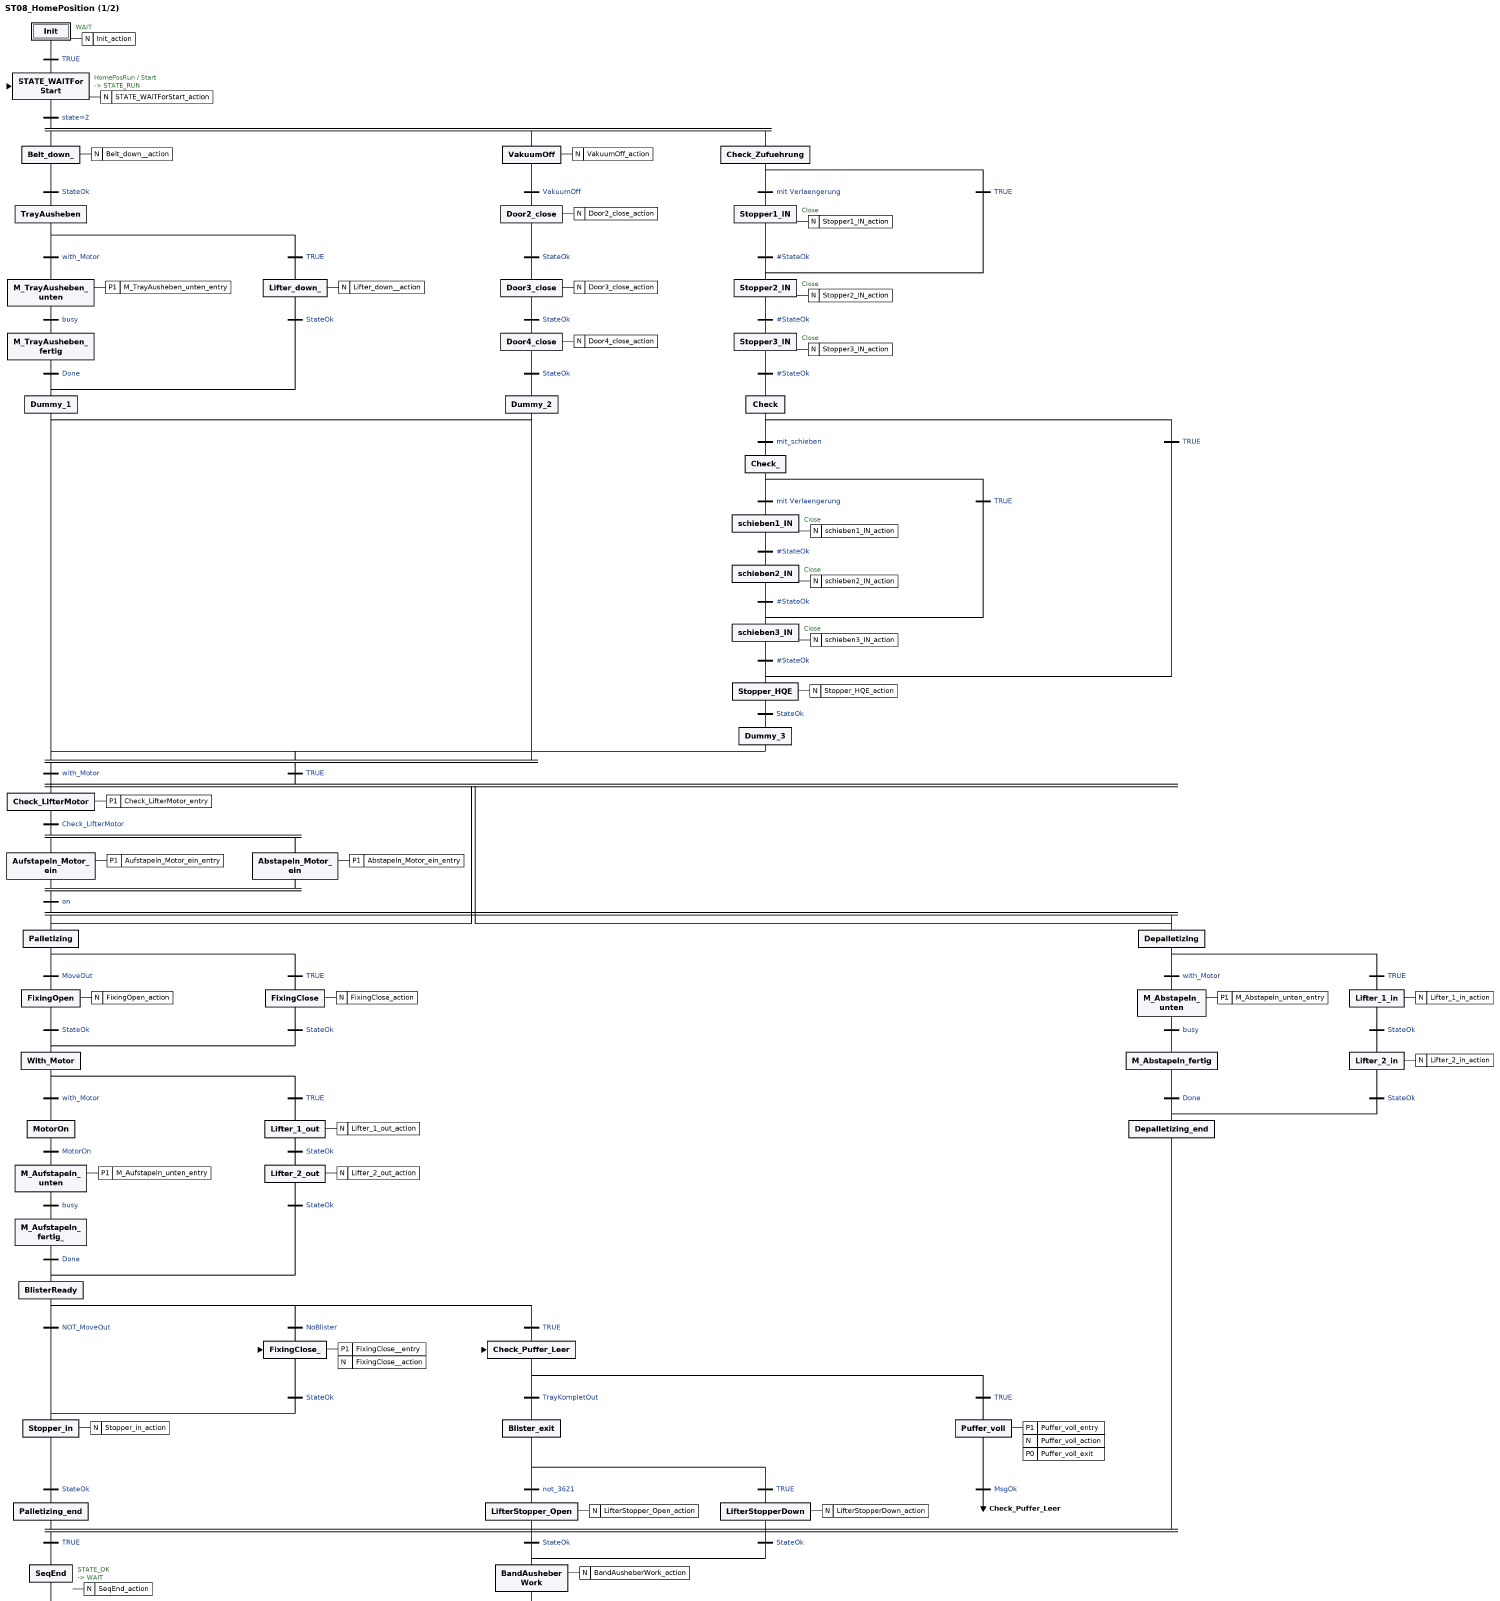
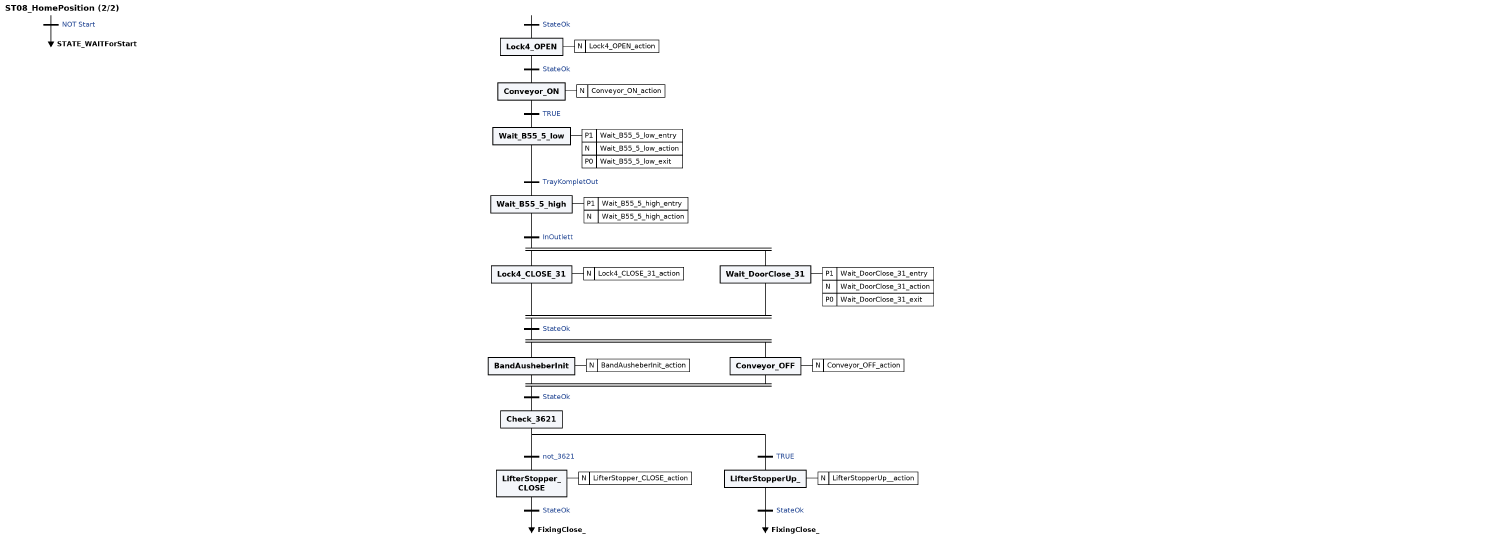
INITIAL_STEP Init: (* WAIT *)
	Init_action(N);
END_STEP
TRANSITION FROM Init TO STATE_WAITForStart := TRUE;
END_TRANSITION
STEP STATE_WAITForStart: (* HomePosRun / Start / -> STATE_RUN *)
	STATE_WAITForStart_action(N);
END_STEP
TRANSITION FROM STATE_WAITForStart TO (Belt_down_, VakuumOff, Check_Zufuehrung) := state=2;
END_TRANSITION
STEP Belt_down_:
	Belt_down__action(N);
END_STEP
TRANSITION FROM Belt_down_ TO TrayAusheben := StateOk;
END_TRANSITION
STEP TrayAusheben:
END_STEP
TRANSITION FROM TrayAusheben TO M_TrayAusheben_unten := with_Motor;
END_TRANSITION
TRANSITION FROM TrayAusheben TO Lifter_down_ := TRUE;
END_TRANSITION
STEP M_TrayAusheben_unten:
	M_TrayAusheben_unten_entry(P1);
END_STEP
TRANSITION FROM M_TrayAusheben_unten TO M_TrayAusheben_fertig := busy;
END_TRANSITION
STEP M_TrayAusheben_fertig:
END_STEP
TRANSITION FROM M_TrayAusheben_fertig TO Dummy_1 := Done;
END_TRANSITION
STEP Lifter_down_:
	Lifter_down__action(N);
END_STEP
TRANSITION FROM Lifter_down_ TO Dummy_1 := StateOk;
END_TRANSITION
STEP Dummy_1:
END_STEP
STEP VakuumOff:
	VakuumOff_action(N);
END_STEP
TRANSITION FROM VakuumOff TO Door2_close := VakuumOff;
END_TRANSITION
STEP Door2_close:
	Door2_close_action(N);
END_STEP
TRANSITION FROM Door2_close TO Door3_close := StateOk;
END_TRANSITION
STEP Door3_close:
	Door3_close_action(N);
END_STEP
TRANSITION FROM Door3_close TO Door4_close := StateOk;
END_TRANSITION
STEP Door4_close:
	Door4_close_action(N);
END_STEP
TRANSITION FROM Door4_close TO Dummy_2 := StateOk;
END_TRANSITION
STEP Dummy_2:
END_STEP
STEP Check_Zufuehrung:
END_STEP
TRANSITION FROM Check_Zufuehrung TO Stopper1_IN := mit Verlaengerung;
END_TRANSITION
TRANSITION FROM Check_Zufuehrung TO Stopper2_IN := TRUE;
END_TRANSITION
STEP Stopper1_IN: (* Close *)
	Stopper1_IN_action(N);
END_STEP
TRANSITION FROM Stopper1_IN TO Stopper2_IN := #StateOk;
END_TRANSITION
STEP Stopper2_IN: (* Close *)
	Stopper2_IN_action(N);
END_STEP
TRANSITION FROM Stopper2_IN TO Stopper3_IN := #StateOk;
END_TRANSITION
STEP Stopper3_IN: (* Close *)
	Stopper3_IN_action(N);
END_STEP
TRANSITION FROM Stopper3_IN TO Check := #StateOk;
END_TRANSITION
STEP Check:
END_STEP
TRANSITION FROM Check TO Check_ := mit_schieben;
END_TRANSITION
TRANSITION FROM Check TO Stopper_HQE := TRUE;
END_TRANSITION
STEP Check_:
END_STEP
TRANSITION FROM Check_ TO schieben1_IN := mit Verlaengerung;
END_TRANSITION
TRANSITION FROM Check_ TO schieben3_IN := TRUE;
END_TRANSITION
STEP schieben1_IN: (* Close *)
	schieben1_IN_action(N);
END_STEP
TRANSITION FROM schieben1_IN TO schieben2_IN := #StateOk;
END_TRANSITION
STEP schieben2_IN: (* Close *)
	schieben2_IN_action(N);
END_STEP
TRANSITION FROM schieben2_IN TO schieben3_IN := #StateOk;
END_TRANSITION
STEP schieben3_IN: (* Close *)
	schieben3_IN_action(N);
END_STEP
TRANSITION FROM schieben3_IN TO Stopper_HQE := #StateOk;
END_TRANSITION
STEP Stopper_HQE:
	Stopper_HQE_action(N);
END_STEP
TRANSITION FROM Stopper_HQE TO Dummy_3 := StateOk;
END_TRANSITION
STEP Dummy_3:
END_STEP
TRANSITION FROM (Dummy_1, Dummy_2, Dummy_3) TO Check_LifterMotor := with_Motor;
END_TRANSITION
TRANSITION FROM (Dummy_1, Dummy_2, Dummy_3) TO (Palletizing, Depalletizing) := TRUE;
END_TRANSITION
STEP Check_LifterMotor:
	Check_LifterMotor_entry(P1);
END_STEP
TRANSITION FROM Check_LifterMotor TO (Aufstapeln_Motor_ein, Abstapeln_Motor_ein) := Check_LifterMotor;
END_TRANSITION
STEP Aufstapeln_Motor_ein:
	Aufstapeln_Motor_ein_entry(P1);
END_STEP
STEP Abstapeln_Motor_ein:
	Abstapeln_Motor_ein_entry(P1);
END_STEP
TRANSITION FROM (Aufstapeln_Motor_ein, Abstapeln_Motor_ein) TO (Palletizing, Depalletizing) := on;
END_TRANSITION
STEP Palletizing:
END_STEP
TRANSITION FROM Palletizing TO FixingOpen := MoveOut;
END_TRANSITION
TRANSITION FROM Palletizing TO FixingClose := TRUE;
END_TRANSITION
STEP FixingOpen:
	FixingOpen_action(N);
END_STEP
TRANSITION FROM FixingOpen TO With_Motor := StateOk;
END_TRANSITION
STEP FixingClose:
	FixingClose_action(N);
END_STEP
TRANSITION FROM FixingClose TO With_Motor := StateOk;
END_TRANSITION
STEP With_Motor:
END_STEP
TRANSITION FROM With_Motor TO MotorOn := with_Motor;
END_TRANSITION
TRANSITION FROM With_Motor TO Lifter_1_out := TRUE;
END_TRANSITION
STEP MotorOn:
END_STEP
TRANSITION FROM MotorOn TO M_Aufstapeln_unten := MotorOn;
END_TRANSITION
STEP M_Aufstapeln_unten:
	M_Aufstapeln_unten_entry(P1);
END_STEP
TRANSITION FROM M_Aufstapeln_unten TO M_Aufstapeln_fertig_ := busy;
END_TRANSITION
STEP M_Aufstapeln_fertig_:
END_STEP
TRANSITION FROM M_Aufstapeln_fertig_ TO BlisterReady := Done;
END_TRANSITION
STEP Lifter_1_out:
	Lifter_1_out_action(N);
END_STEP
TRANSITION FROM Lifter_1_out TO Lifter_2_out := StateOk;
END_TRANSITION
STEP Lifter_2_out:
	Lifter_2_out_action(N);
END_STEP
TRANSITION FROM Lifter_2_out TO BlisterReady := StateOk;
END_TRANSITION
STEP BlisterReady:
END_STEP
TRANSITION FROM BlisterReady TO Stopper_in := NOT_MoveOut;
END_TRANSITION
TRANSITION FROM BlisterReady TO FixingClose_ := NoBlister;
END_TRANSITION
TRANSITION FROM BlisterReady TO Check_Puffer_Leer := TRUE;
END_TRANSITION
STEP FixingClose_:
	FixingClose__entry(P1);
	FixingClose__action(N);
END_STEP
TRANSITION FROM FixingClose_ TO Stopper_in := StateOk;
END_TRANSITION
STEP Check_Puffer_Leer:
END_STEP
TRANSITION FROM Check_Puffer_Leer TO Blister_exit := TrayKompletOut;
END_TRANSITION
TRANSITION FROM Check_Puffer_Leer TO Puffer_voll := TRUE;
END_TRANSITION
STEP Puffer_voll:
	Puffer_voll_entry(P1);
	Puffer_voll_action(N);
	Puffer_voll_exit(P0);
END_STEP
TRANSITION FROM Puffer_voll TO Check_Puffer_Leer := MsgOk;
END_TRANSITION
STEP Blister_exit:
END_STEP
TRANSITION FROM Blister_exit TO LifterStopper_Open := not_3621;
END_TRANSITION
TRANSITION FROM Blister_exit TO LifterStopperDown := TRUE;
END_TRANSITION
STEP LifterStopper_Open:
	LifterStopper_Open_action(N);
END_STEP
TRANSITION FROM LifterStopper_Open TO BandAusheberWork := StateOk;
END_TRANSITION
STEP LifterStopperDown:
	LifterStopperDown_action(N);
END_STEP
TRANSITION FROM LifterStopperDown TO BandAusheberWork := StateOk;
END_TRANSITION
STEP BandAusheberWork:
	BandAusheberWork_action(N);
END_STEP
TRANSITION FROM BandAusheberWork TO Lock4_OPEN := StateOk;
END_TRANSITION
STEP Lock4_OPEN:
	Lock4_OPEN_action(N);
END_STEP
TRANSITION FROM Lock4_OPEN TO Conveyor_ON := StateOk;
END_TRANSITION
STEP Conveyor_ON:
	Conveyor_ON_action(N);
END_STEP
TRANSITION FROM Conveyor_ON TO Wait_B55_5_low := TRUE;
END_TRANSITION
STEP Wait_B55_5_low:
	Wait_B55_5_low_entry(P1);
	Wait_B55_5_low_action(N);
	Wait_B55_5_low_exit(P0);
END_STEP
TRANSITION FROM Wait_B55_5_low TO Wait_B55_5_high := TrayKompletOut;
END_TRANSITION
STEP Wait_B55_5_high:
	Wait_B55_5_high_entry(P1);
	Wait_B55_5_high_action(N);
END_STEP
TRANSITION FROM Wait_B55_5_high TO (Lock4_CLOSE_31, Wait_DoorClose_31) := InOutlett;
END_TRANSITION
STEP Lock4_CLOSE_31:
	Lock4_CLOSE_31_action(N);
END_STEP
STEP Wait_DoorClose_31:
	Wait_DoorClose_31_entry(P1);
	Wait_DoorClose_31_action(N);
	Wait_DoorClose_31_exit(P0);
END_STEP
TRANSITION FROM (Lock4_CLOSE_31, Wait_DoorClose_31) TO (BandAusheberInit, Conveyor_OFF) := StateOk;
END_TRANSITION
STEP BandAusheberInit:
	BandAusheberInit_action(N);
END_STEP
STEP Conveyor_OFF:
	Conveyor_OFF_action(N);
END_STEP
TRANSITION FROM (BandAusheberInit, Conveyor_OFF) TO Check_3621 := StateOk;
END_TRANSITION
STEP Check_3621:
END_STEP
TRANSITION FROM Check_3621 TO LifterStopper_CLOSE := not_3621;
END_TRANSITION
TRANSITION FROM Check_3621 TO LifterStopperUp_ := TRUE;
END_TRANSITION
STEP LifterStopper_CLOSE:
	LifterStopper_CLOSE_action(N);
END_STEP
TRANSITION FROM LifterStopper_CLOSE TO FixingClose_ := StateOk;
END_TRANSITION
STEP LifterStopperUp_:
	LifterStopperUp__action(N);
END_STEP
TRANSITION FROM LifterStopperUp_ TO FixingClose_ := StateOk;
END_TRANSITION
STEP Stopper_in:
	Stopper_in_action(N);
END_STEP
TRANSITION FROM Stopper_in TO Palletizing_end := StateOk;
END_TRANSITION
STEP Palletizing_end:
END_STEP
STEP Depalletizing:
END_STEP
TRANSITION FROM Depalletizing TO M_Abstapeln_unten := with_Motor;
END_TRANSITION
TRANSITION FROM Depalletizing TO Lifter_1_in := TRUE;
END_TRANSITION
STEP M_Abstapeln_unten:
	M_Abstapeln_unten_entry(P1);
END_STEP
TRANSITION FROM M_Abstapeln_unten TO M_Abstapeln_fertig := busy;
END_TRANSITION
STEP M_Abstapeln_fertig:
END_STEP
TRANSITION FROM M_Abstapeln_fertig TO Depalletizing_end := Done;
END_TRANSITION
STEP Lifter_1_in:
	Lifter_1_in_action(N);
END_STEP
TRANSITION FROM Lifter_1_in TO Lifter_2_in := StateOk;
END_TRANSITION
STEP Lifter_2_in:
	Lifter_2_in_action(N);
END_STEP
TRANSITION FROM Lifter_2_in TO Depalletizing_end := StateOk;
END_TRANSITION
STEP Depalletizing_end:
END_STEP
TRANSITION FROM (Palletizing_end, Depalletizing_end) TO SeqEnd := TRUE;
END_TRANSITION
STEP SeqEnd: (* STATE_OK / -> WAIT *)
	SeqEnd_action(N);
END_STEP
TRANSITION FROM SeqEnd TO STATE_WAITForStart := NOT Start;
END_TRANSITION

ACTION Init_action:
Start:=FALSE;
State:=STATE_WAIT;
END_ACTION

ACTION STATE_WAITForStart_action:
IF	Start THEN
	State:=STATE_RUN;
	Result:=RESULT_NON;
	SFCTimeStart:=TIME();
END_IF
END_ACTION

ACTION Belt_down__action:
ST08_404_Y52_0.MoveInit:=TRUE;
END_ACTION

ACTION M_TrayAusheben_unten_entry:
ST08_190_M1.MoveAbs:=TRUE;
ST08_190_M1.Vorgabe_Pos_Abs:=TD.PosTrayAusheben[1].Pos;	(*1=unten, 2=oben, *)
END_ACTION

ACTION Lifter_down__action:
ST08_406_Y52_3.MoveInit:=TRUE;
END_ACTION

ACTION VakuumOff_action:
ST08_403_Y50_6.MoveInit := TRUE;
ST08_403_Y50_7.MoveInit := TRUE;
END_ACTION

ACTION Door2_close_action:
ST08_405_Y51_0.MoveInit:=TRUE;
END_ACTION

ACTION Door3_close_action:
ST08_406_Y51_2.MoveInit:=TRUE;
END_ACTION

ACTION Door4_close_action:
ST08_407_Y51_4.MoveInit:=TRUE;
END_ACTION

ACTION Stopper1_IN_action:
ST08_400_Y50_0.MoveInit:=TRUE; (* Stopper Traystapel Einlaufb. hinten links + rechts AST (Valve) *)
END_ACTION

ACTION Stopper2_IN_action:
ST08_400_Y50_2.MoveInit:=TRUE;
END_ACTION

ACTION Stopper3_IN_action:
ST08_402_Y50_4.MoveInit:=TRUE;
END_ACTION

ACTION schieben1_IN_action:
ST08_401_Y52_4.MoveInit:=TRUE; (*  Traystapel schieben hinten AST (Valve) *)
END_ACTION

ACTION schieben2_IN_action:
ST08_402_Y52_6.MoveInit:=TRUE;
END_ACTION

ACTION schieben3_IN_action:
ST08_402_Y52_7.MoveInit:=TRUE;
END_ACTION

ACTION Stopper_HQE_action:
ST08_404_Y51_6.MoveInit:=TRUE;
END_ACTION

ACTION Check_LifterMotor_entry:
ST08_180_M1.MotorOn:=NOT ST08_180_M1.On;
ST08_185_M1.MotorOn:=NOT ST08_185_M1.On;
END_ACTION

ACTION Aufstapeln_Motor_ein_entry:
ST08_185_M1.Vorgabe_Velo:=1750;
END_ACTION

ACTION Abstapeln_Motor_ein_entry:
ST08_180_M1.Vorgabe_Velo:=1750;
END_ACTION

ACTION FixingOpen_action:
ST08_408_Y54_0.MoveWork:=TRUE;
END_ACTION

ACTION FixingClose_action:
ST08_408_Y54_0.MoveInit:=TRUE;
END_ACTION

ACTION M_Aufstapeln_unten_entry:
ST08_185_M1.MoveAbs:=TRUE;
ST08_185_M1.Vorgabe_Pos_Abs:=TD.PosAufstapeln[1].Pos;	(*1=unten, 2= mitte, 3=oben, 4=frei*)
END_ACTION

ACTION Lifter_1_out_action:
ST08_408_Y54_2.MoveInit:=TRUE;
END_ACTION

ACTION Lifter_2_out_action:
ST08_408_Y54_4.MoveInit:=TRUE;
END_ACTION

ACTION FixingClose__entry:
MP.ST08.NoOfBlisterInStackerOut:=0;
END_ACTION

ACTION FixingClose__action:
ST08_408_Y54_0.MoveInit:=TRUE;
END_ACTION

ACTION Puffer_voll_entry:
MessageHandler.ClearMessageLines(sVisu:=Visu.Message);
END_ACTION

ACTION Puffer_voll_action:
MessageHandler.Msg.ID:='PM201';
MessageHandler.Msg.Name:='St08 Stau im Auslauf';
MessageHandler.Msg.Text:='Auslaufand voll!! Blister entnehmen!!';
MessageHandler.Msg.Color:=Color.blue;
MessageHandler.Msg.Station:=0;


MessageHandler(
	Prio:=2, 							(*1=highest, .. , 4=lowest*)
	Btn1Addr:=ADR(MsgOk),			(*Address of Button1 , if Zero then Button is unvisible*)
	Btn2Addr:=,			(*Address of Button2 , if Zero then Button is unvisible*)
	sVisu:=Visu.Message);
END_ACTION

ACTION Puffer_voll_exit:
MsgOk:=FALSE;
MsgCancel:=FALSE;
END_ACTION

ACTION LifterStopper_Open_action:
ST08_400_Y52_5.MoveWork :=TRUE;
END_ACTION

ACTION LifterStopperDown_action:
ST08_408_Y54_4.MoveInit:=TRUE;
END_ACTION

ACTION BandAusheberWork_action:
ST08_404_Y52_0.MoveWork:=TRUE;
END_ACTION

ACTION Lock4_OPEN_action:
ST08_407_Y51_4.MoveWork:=TRUE;
END_ACTION

ACTION Conveyor_ON_action:
ST08_Palletizing.ConveyorOn:=TRUE;
END_ACTION

ACTION Wait_B55_5_low_entry:
ProcessMessage01:='';
END_ACTION

ACTION Wait_B55_5_low_action:
ProcessMessage01:='1IM12';(*'St. 8 warte Tray ausgelaufen*)
END_ACTION

ACTION Wait_B55_5_low_exit:
ProcessMessage01:='';
END_ACTION

ACTION Wait_B55_5_high_entry:
ProcessMessage01:='';
END_ACTION

ACTION Wait_B55_5_high_action:
ProcessMessage01:='1IM13';(*St. 8 warte Tray auf Rollenbahn*)
END_ACTION

ACTION Lock4_CLOSE_31_action:
ST08_407_Y51_4.MoveInit:=TRUE;
END_ACTION

ACTION Wait_DoorClose_31_entry:
ProcessMessage01:='';
END_ACTION

ACTION Wait_DoorClose_31_action:
ProcessMessage01:='1IM14';(*'St.8 warte Türe 4 auslauf geschlossen*)
END_ACTION

ACTION Wait_DoorClose_31_exit:
ProcessMessage01:='';
END_ACTION

ACTION BandAusheberInit_action:
ST08_404_Y52_0.MoveInit:=TRUE;
END_ACTION

ACTION Conveyor_OFF_action:
ST08_Palletizing.ConveyorOn:=FALSE;
END_ACTION

ACTION LifterStopper_CLOSE_action:
ST08_400_Y52_5.MoveInit:=TRUE;
END_ACTION

ACTION LifterStopperUp__action:
ST08_408_Y54_4.MoveWork:=TRUE;
END_ACTION

ACTION Stopper_in_action:
ST08_400_Y52_5.MoveWork:=TRUE;
END_ACTION

ACTION M_Abstapeln_unten_entry:
ST08_180_M1.MoveAbs:=TRUE;
ST08_180_M1.Vorgabe_Pos_Abs:=TD.PosAbstapeln[1].Pos;	(*1=unten, 2= mitte, 3=oben, 4=frei*)
END_ACTION

ACTION Lifter_1_in_action:
ST08_404_Y53_0.MoveInit:=TRUE;
END_ACTION

ACTION Lifter_2_in_action:
ST08_404_Y53_2.MoveInit:=TRUE;
END_ACTION

ACTION SeqEnd_action:
IF	ST08_406_B54_3.BitInToCheck THEN
	ST08_CallPRGs.PosIdxHelp:=0;
END_IF

IF 	State=STATE_RUN THEN
	SFCTime:=TIME_TO_DINT(TIME()-SFCTimeStart);
	State:=STATE_OK;
END_IF

IF 	NOT Start THEN
	State:=STATE_WAIT;
END_IF
END_ACTION

TRANSITION StateOk:
ST08_404_Y52_0.State=STATE_OK
END_TRANSITION

TRANSITION with_Motor:
MP.ST08.TrayAushebenMotor
END_TRANSITION

TRANSITION busy:
ST08_190_M1.Busy
END_TRANSITION

TRANSITION Done:
ST08_190_M1.Done
END_TRANSITION

TRANSITION StateOk:
ST08_406_Y52_3.State=STATE_OK
END_TRANSITION

TRANSITION VakuumOff:
ST08_403_Y50_6.State=STATE_OK AND
ST08_403_Y50_7.State=STATE_OK
END_TRANSITION

TRANSITION StateOk:
ST08_405_Y51_0.State=STATE_OK
END_TRANSITION

TRANSITION StateOk:
ST08_406_Y51_2.State=STATE_OK
END_TRANSITION

TRANSITION StateOk:
ST08_407_Y51_4.State=STATE_OK
END_TRANSITION

TRANSITION mit Verlaengerung:
MP.ST08.Trayzufuhr_Verlaengerung
END_TRANSITION

TRANSITION #StateOk:
ST08_400_Y50_0.State=STATE_OK
END_TRANSITION

TRANSITION #StateOk:
ST08_400_Y50_2.State=STATE_OK
END_TRANSITION

TRANSITION #StateOk:
ST08_402_Y50_4.State=STATE_OK
END_TRANSITION

TRANSITION mit_schieben:
MP.ST08.Traystapel_schieben
END_TRANSITION

TRANSITION mit Verlaengerung:
MP.ST08.Trayzufuhr_Verlaengerung
END_TRANSITION

TRANSITION #StateOk:
ST08_401_Y52_4.State=STATE_OK
END_TRANSITION

TRANSITION #StateOk:
ST08_402_Y52_6.State=STATE_OK
END_TRANSITION

TRANSITION #StateOk:
ST08_402_Y52_7.State=STATE_OK
END_TRANSITION

TRANSITION StateOk:
ST08_404_Y51_6.State=STATE_OK
END_TRANSITION

TRANSITION with_Motor:
MP.ST08.StapelMotor
END_TRANSITION

TRANSITION Check_LifterMotor:
NOT ST08_180_M1.Error_ AND
ST08_180_M1.On AND
NOT ST08_185_M1.Error_ AND
ST08_185_M1.On
END_TRANSITION

TRANSITION on:
ST08_180_M1.on AND
ST08_185_M1.on
END_TRANSITION

TRANSITION MoveOut:
ST08_Palletizing.MoveOut
END_TRANSITION

TRANSITION StateOk:
ST08_408_Y54_0.State=STATE_OK
END_TRANSITION

TRANSITION StateOk:
ST08_408_Y54_0.State=STATE_OK
END_TRANSITION

TRANSITION with_Motor:
MP.ST08.StapelMotor
END_TRANSITION

TRANSITION MotorOn:
ST08_185_M1.On
END_TRANSITION

TRANSITION busy:
ST08_185_M1.Busy
END_TRANSITION

TRANSITION Done:
ST08_185_M1.Done
END_TRANSITION

TRANSITION StateOk:
ST08_408_Y54_2.State=STATE_OK
END_TRANSITION

TRANSITION StateOk:
ST08_408_Y54_4.State=STATE_OK
END_TRANSITION

TRANSITION NOT_MoveOut:
NOT ST08_Palletizing.MoveOut
END_TRANSITION

TRANSITION NoBlister:
ST08_407_B55_4.BitInToCheck (* Tray in Aufstapelposition eingelaufen STN8 *)
END_TRANSITION

TRANSITION StateOk:
ST08_408_Y54_0.State=STATE_OK
END_TRANSITION

TRANSITION TrayKompletOut:
ST08_409_B55_5.BitInToCheck
END_TRANSITION

TRANSITION not_3621:
NOT MP.ST03.SGM_3621
END_TRANSITION

TRANSITION StateOk:
(*ST08_408_Y54_4.State=STATE_OK*)

ST08_400_Y52_5.State=STATE_OK AND
gTipImp
END_TRANSITION

TRANSITION StateOk:
ST08_408_Y54_4.State =STATE_OK AND
gTipImp
END_TRANSITION

TRANSITION StateOk:
(*ST08_408_Y54_4.State=STATE_OK*)

ST08_400_Y52_5.State=STATE_OK AND
gTipImp
END_TRANSITION

TRANSITION StateOk:
ST08_407_Y51_4.State=STATE_OK AND
gTipImp
END_TRANSITION

TRANSITION TrayKompletOut:
NOT ST08_409_B55_5.BitInToCheck AND
gTipImp
END_TRANSITION

TRANSITION InOutlett:
ST08_409_B55_5.BitInToCheck AND
gTipImp
END_TRANSITION

TRANSITION StateOk:
ST08_407_Y51_4.State=STATE_OK AND
NOT ST00_227_S2.BitInToCheck AND
NOT ST00_230_S1.BitInToCheck AND
gTipImp
END_TRANSITION

TRANSITION StateOk:
ST08_404_Y52_0.State=STATE_OK
END_TRANSITION

TRANSITION not_3621:
NOT MP.ST03.SGM_3621
END_TRANSITION

TRANSITION StateOk:
(*ST08_408_Y54_4.State=STATE_OK*)

ST08_400_Y52_5.State=STATE_OK AND
gTipImp
END_TRANSITION

TRANSITION StateOk:
ST08_408_Y54_4.State=STATE_OK

AND gTipImp
END_TRANSITION

TRANSITION StateOk:
(*ST08_408_Y54_4.State=STATE_OK*)

ST08_400_Y52_5.State=STATE_OK
OR
MP.ST03.SGM_3621
END_TRANSITION

TRANSITION with_Motor:
MP.ST08.StapelMotor
END_TRANSITION

TRANSITION busy:
ST08_180_M1.Busy
END_TRANSITION

TRANSITION Done:
ST08_180_M1.Done
END_TRANSITION

TRANSITION StateOk:
ST08_404_Y53_0.State=STATE_OK
END_TRANSITION

TRANSITION StateOk:
 ST08_404_Y53_2.State=STATE_OK
END_TRANSITION
END_PROGRAM

(* POU System/GeneralFunctions/CallGeneralFunctions, ST *)
PROGRAM CallGeneralFunctions
VAR
	gFB_GETLOCALSYSTEMTIME		:	FB_LocalSystemTime;

	SetLocalTime			: 	NT_SetLocalTime;
	SetTimeStruct			:		TIMESTRUCT;
	SetTimePicEnabled		: 	R_TRIG;

	GetLocalAmsNetId		: 	FB_GetLocalAmsNetId;
	FBWritePersistentData	:	WritePersistentData;

	VisuShutDown:NT_Shutdown;

	TonVisuShutDown : TON;
	ShutDownManual:BOOL;
	ExecuteEverySecondAdFirstCycle: BOOL;
	FBSwitchToConfigMode:TC_Config;
	SwitchToConfigMode: BOOL;

	SavePersistentData: BOOL;
	TDValid								:	R_TRIG;
	PDValid								:	R_TRIG;
	wYear: WORD;
	wMonth: WORD;
	wDay: WORD;
	wHour: WORD;
	wMin: WORD;
	wSec: WORD;

(* Generate Pulses *)
	Pulse1000ms					:	GEN_PULSE;
	Pulse0500ms					:	GEN_PULSE;
	Pulse0100ms					:	GEN_PULSE;
	Pulse0050ms					:	GEN_PULSE;
	Pulse0025ms					:	GEN_PULSE;

	PersDatenCopy					:sPersDaten;

END_VAR
ExecuteEverySecondAdFirstCycle:=SystemTaskInfoArr[SystemInfo.runTimeNo].firstCycle;

GetLocalAmsNetId(
	bExecute:= ExecuteEverySecondAdFirstCycle,
	tTimeout:= t#1s,
	AddrString=> LocalAmsNetIdStr,
	AddrBytes=> LocalAmsNetIdArr);

FBSwitchToConfigMode(
	NETID:= LocalAmsNetIdStr,
	SET:= SwitchToConfigMode ,
	TMOUT:=t#10s );


TDValid(CLK:=gTypeDataValid );

(*Schreibe bei einer Änderung*)
PDValid(CLK:=
	(MEMCMP(ADR(PersDatenCopy), ADR(PersDaten), SIZEOF(PersDatenCopy)) <> 0 ) AND
	ModeSelect.Mode <= MODE_AUTO_RUN);

SavePersistentData:=  TDValid.Q OR PDValid.Q OR visu.SavePersistentData;


FBWritePersistentData(
	NETID:='' ,
	PORT:= 801,
	START:= SavePersistentData,
	TMOUT:=t#2000ms );

visu.SavePersistentData:=FALSE;

(*Impuls Generieren*)
Pulse1000ms(ENQ:=TRUE , PTH:=t#1s, 		PTL:= t#1s, 		Q=>vGlbImpuls_1000ms );
Pulse0500ms(ENQ:=TRUE , PTH:=t#500ms, PTL:= t#500ms, 	Q=>vGlbImpuls_0500ms );
Pulse0100ms(ENQ:=TRUE , PTH:=t#100ms, PTL:= t#100ms, 	Q=>vGlbImpuls_0100ms );
Pulse0050ms(ENQ:=TRUE , PTH:=t#50ms, PTL:= t#50ms, 	Q=>vGlbImpuls_0050ms );
Pulse0025ms(ENQ:=TRUE , PTH:=t#25ms, PTL:= t#25ms, 	Q=>vGlbImpuls_0025ms );


(*		Shutdown Visu on USV - Alarm *)

TonVisuShutDown(IN:= ShutDownManual , PT:= t#2s );

VisuShutDown(
	NETID:= '' ,
	DELAY:=3 ,
	START:= TonVisuShutDown.Q,
	TMOUT:=t#20s );

gFB_GETLOCALSYSTEMTIME(
	sNetID:='' ,
	bEnable:=TRUE ,
	dwCycle:=1 );

gVarStrSystemTime:=SYSTEMTIME_TO_STRING(gFB_GETLOCALSYSTEMTIME.systemTime);
gVarDTSystemtime:=SYSTEMTIME_TO_DT(gFB_GETLOCALSYSTEMTIME.SystemTime);
gVarSystemtime:=gFB_GETLOCALSYSTEMTIME.systemTime;

wYear:=gVarSystemtime.wYear;
wMonth:=gVarSystemtime.wMonth;
wDay:=gVarSystemtime.wDay;
wHour:=gVarSystemtime.wHour;
wMin:=gVarSystemtime.wMinute;
wSec:=gVarSystemtime.wSecond;
gVarStrSystemTime:='';
IF 	wDay<10 THEN
	gVarStrSystemTime:=CONCAT(gVarStrSystemTime ,WORD_TO_STRING(0));
END_IF
gVarStrSystemTime:=CONCAT(gVarStrSystemTime ,WORD_TO_STRING(wDay));
gVarStrSystemTime:=CONCAT(gVarStrSystemTime , '.');
IF 	wMonth<10 THEN
	gVarStrSystemTime:=CONCAT(gVarStrSystemTime ,WORD_TO_STRING(0));
END_IF
gVarStrSystemTime:=CONCAT(gVarStrSystemTime ,WORD_TO_STRING(wMonth));
gVarStrSystemTime:=CONCAT(gVarStrSystemTime , '.');
gVarStrSystemTime:=CONCAT(gVarStrSystemTime ,WORD_TO_STRING(wYear));

gVarStrSystemTime:=CONCAT(gVarStrSystemTime , ' ');
IF 	wHour<10 THEN
	gVarStrSystemTime:=CONCAT(gVarStrSystemTime ,WORD_TO_STRING(0));
END_IF
gVarStrSystemTime:=CONCAT(gVarStrSystemTime ,WORD_TO_STRING(wHour));
gVarStrSystemTime:=CONCAT(gVarStrSystemTime , ':');
IF 	wMin<10 THEN
	gVarStrSystemTime:=CONCAT(gVarStrSystemTime ,WORD_TO_STRING(0));
END_IF
gVarStrSystemTime:=CONCAT(gVarStrSystemTime ,WORD_TO_STRING(wMin));
gVarStrSystemTime:=CONCAT(gVarStrSystemTime , ':');
IF 	wSec<10 THEN
	gVarStrSystemTime:=CONCAT(gVarStrSystemTime ,WORD_TO_STRING(0));
END_IF
gVarStrSystemTime:=CONCAT(gVarStrSystemTime ,WORD_TO_STRING(wSec));

SetTimePicEnabled(CLK:= currentVisu='MP_DATE' );

IF 	SetTimePicEnabled.Q THEN
	SetTimeStruct:=gVarSystemtime;
END_IF

SetLocalTime(
	NETID:= '',
	TIMESTR:= SetTimeStruct,
	TMOUT:= t#10s);
END_PROGRAM

(* POU System/HelpFunctions/GEN_PULSE, ST *)
FUNCTION_BLOCK GEN_PULSE
VAR_INPUT
	ENQ 		: BOOL := TRUE;
	PTH 		:TIME;
	PTL 		:TIME;
END_VAR
VAR_OUTPUT
	Q 			:BOOL;
	Q_FP		:BOOL;
END_VAR
VAR
	ein			:TIME;
	aus			:TIME;
	cyc			:TIME;
	init			:BOOL;
	Q_RTRIG	:R_TRIG;
END_VAR

(*GEN_PULSE uses the internal sps timer to generate a continuous output waveform with programmable high and low time.
the accuracy of gen_pulse is depending on the system timer.
when time is 0 the high and low times are exactly one cycle.
ENQ = TRUE will start and ENQ = FALSE will stop the generator.*)
(* read system timer *)
cyc:=DWORD_TO_TIME(SystemTaskInfoArr[SystemInfo.runTimeNo].cycleTime/10000);
IF 	NOT init THEN
	init:=TRUE;
	aus:=t#0s;
	ein:=t#0s;

END_IF;
IF 	enq AND init THEN
	IF ein<= pth THEN
		ein:=ein+cyc;
		q:=TRUE;
	ELSE
		q:=FALSE;
		aus:=aus+cyc;
		IF 	aus>=ptl THEN
			init:=FALSE;
		END_IF;
	END_IF;

ELSE
	Q := FALSE;
END_IF;

Q_RTRIG(CLK:=Q , Q=>Q_FP );
END_FUNCTION_BLOCK

(* POU zLibrary/ept/Programmbausteine/ST_UPS, ST *)
PROGRAM ST_UPS
VAR_INPUT
	b_Ups				: BOOL;
END_VAR
VAR_IN_OUT

END_VAR
VAR_OUTPUT
END_VAR
VAR
	fb_state_entry		: ST_StateEntry;

	nLastErrID			: UDINT;

	fbGetUpsStatus		: FB_GetUPSStatus;

	bm_ReplaceBattery 	: BOOL;
	bm_NoPower 		: BOOL;
	bm_StatusNotValid 	: BOOL;
	bm_Check			: BOOL;
	fb_rTrig_ReplaceBattery 	: R_TRIG;
	fb_rTrig_NoPower 		: R_TRIG;
	fb_rTrig_StatusNotValid 	: R_TRIG;
	fb_rTrig_Check 			: R_TRIG;
	fb_rTrig_Reset			: R_TRIG;

	bmError				: ErrorStruct;

	FB_ReadXmlLineMsg		:FB_ReadXmlLine;
	tmpErrorText				:STRING;

END_VAR
(*======================================================
   ST: ST_UPS
 ------------------------------------------------------
   Auth: 	Thomas Vilgis    						 
   Date: 	21.06.2018    						     
   Rev.: 		1.0	
   Desc:		Der Baustein liest den Status des Akkupacks aus.
			Die restliche Akkulaufzeit in Minuten kann abgefragt werden.
			Wenn der Akkupack getauscht werden muss wird angezeigt.
			Wenn sich der PC im Netzbetrieb befindet wird angezeigt.
   Historie: 	1.0

 ========================================================*)

fb_state_entry(	i16_pos:= 1);

CASE fb_state_entry.i16_step OF
(*=======================================================*)
	INIT_OBJ:

			fb_state_entry.i16_next_step := INIT;


(*=======================================================*)
	INIT:
		IF fb_state_entry.E THEN

			bm_ReplaceBattery := FALSE;
			bm_NoPower := FALSE;
			bm_StatusNotValid := FALSE;
			bm_Check:= FALSE;
			fbGetUpsStatus.bEnable := FALSE;
		END_IF

		(*-----------------------Weiterschaltbedingungen----------------------------*)
		fb_state_entry.i16_next_step := BEREIT;

(*=======================================================*)
	BEREIT:
		IF 	fb_state_entry.E THEN
			;
		END_IF

		fbGetUpsStatus.bEnable := b_Ups;

		(*-----------------------Weiterschaltbedingungen----------------------------*)
		IF b_Ups THEN
			IF 	fbGetUpsStatus.bValid THEN
				fb_state_entry.i16_next_step := 110;
			ELSIF
				fb_state_entry.fb_ton_Step.ET > t#20s THEN
				bm_StatusNotValid := TRUE;
				fb_state_entry.i16_next_step := FEHLER;
			END_IF
		END_IF

		IF 	fb_state_entry.X THEN
			;
		END_IF

(*=======================================================*)
	110:	(* Evaluation *)

		(*-----------------------Weiterschaltbedingungen----------------------------*)
		IF fbGetUpsStatus.bValid THEN
			IF NOT fbGetUpsStatus.bError THEN
				CASE fbGetUpsStatus.stStatus.eBatteryStatus OF
					BatteryUnknownStatus:	(*Der Akkustatus ist unbekannt*)
						;
					BatteryOk:			(*Der Akku ist in Ordnung*)
						bm_ReplaceBattery := FALSE;
					BatteryReplace:		(*Der Akku sollte gewechselt werden*)
						bm_ReplaceBattery := TRUE;
				END_CASE

				CASE fbGetUpsStatus.stStatus.eCommStatus OF
					UpsCommUnknownStatus:	(*Kommunikationsstatus zur USV-Hardware ist unbekannt*)
						;
					UpsCommOk:		(*Kommunikation zur USV-Hardware ist hergestellt*)
						;
					UpsCommFailed:		(*Kommunikation zur USV wurde unterbrochen*)
						;
				END_CASE

				CASE fbGetUpsStatus.stStatus.ePowerStatus OF
					PowerUnknownStatus:	(*Der Status der Stromversorgung ist unbekannt*)
						;
					PowerOnLine:		(*Das Gerät befindet sich im Netzbetrieb*)
						bm_NoPower := FALSE;
					PowerOnBattery:	(*Stromausfall ist aufgetreten und das Gerät befindet sich im Akkubetrieb*)
						bm_NoPower := TRUE;
				END_CASE
			ELSE
				nLastErrID := fbGetUpsStatus.nErrId;
				fb_state_entry.i16_next_step := FEHLER;
			END_IF
		ELSE
			bm_StatusNotValid := TRUE;
			fb_state_entry.i16_next_step := FEHLER;
		END_IF

(*=======================================================*)
	FEHLER:	 fb_state_entry.s_debugtext:=CONCAT('Error ID: ',UDINT_TO_STRING(nLastErrID));

		IF fb_state_entry.E THEN
			fbGetUpsStatus.bEnable := FALSE;
		END_IF

		(*-----------------------Weiterschaltbedingungen----------------------------*)
		IF 	(fb_state_entry.fb_ton_Step.Q  AND bm_StatusNotValid) OR
			gResetAll THEN
			fb_state_entry.i16_next_step := INIT;
		END_IF

END_CASE

fb_state_entry(i16_pos:= 2 );

fbGetUpsStatus(
	sNetId:= ,	(* wenn in AmsNetId nichts drin steht, wird immer die lokale genommen*)
	nPort:= 0,
	bEnable:= ,
	bValid=> ,
	bError=> ,
	nErrId=> ,
	stStatus=> );

(*Checks zurücksetzen*)
fb_rTrig_Reset(CLK:=gResetAll);
IF fb_rTrig_Reset.Q THEN
	CheckBounds_ErrCnt:=0;
	CheckByteZeroDiv_ErrCnt:=0;
	CheckDWordZeroDiv_ErrCnt:=0;
	CheckRealZeroDiv_ErrCnt:=0;
	CheckWordZeroDiv_ErrCnt:=0;
	CheckRangeSigned_ErrCnt:=0;
	CheckRangeUnsigned_ErrCnt:=0;
END_IF

bm_Check:=ABS(
	CheckBounds_ErrCnt+
	CheckByteZeroDiv_ErrCnt+
	CheckDWordZeroDiv_ErrCnt+
	CheckRealZeroDiv_ErrCnt+
	CheckWordZeroDiv_ErrCnt+
	CheckRangeSigned_ErrCnt+
	CheckRangeUnsigned_ErrCnt	)  > 2 ;

(* Generate information Errorlog *)
fb_rTrig_ReplaceBattery(CLK:=bm_ReplaceBattery);
fb_rTrig_NoPower(CLK:=bm_NoPower);
fb_rTrig_StatusNotValid(CLK:=bm_StatusNotValid);
fb_rTrig_Check(CLK:=bm_Check);

IF 	fb_rTrig_ReplaceBattery.Q THEN
	tmpErrorText:='bm_ReplaceBattery';					(*USV Aku defekt! =>tauschen*)
	bmError.DateTime:= gVarDTSystemtime;
END_IF
IF	fb_rTrig_NoPower.Q THEN
	tmpErrorText:='bm_NoPower';						(*Stromausfall Steuerung wird von der USV versorgt!*)
	bmError.DateTime:= gVarDTSystemtime;
END_IF
IF	fb_rTrig_StatusNotValid.Q THEN
	tmpErrorText:='bm_StatusNotValid';					(*USV Status kann nicht ausgelesen werden*)
	bmError.DateTime:= gVarDTSystemtime;
END_IF
IF	fb_rTrig_Check.Q THEN
	tmpErrorText:='bm_Check';							(*Error Check's*)
	bmError.DateTime:= gVarDTSystemtime;
END_IF

IF 	bm_ReplaceBattery OR
	bm_NoPower OR
	bm_StatusNotValid OR
	bm_Check THEN
	bmError.Typ:= 1;										(* 0=red 1:=orange 2:=blue *)
	bmError.No:= 1;
	ErrorHandler.AddError(ErrorToAdd:=bmError,sVisu:=Visu.ErrorHandler);
END_IF

FB_ReadXmlLineMsg(
	Prefix:= 'MSG',
	ID:= tmpErrorText,
	File:= 'MSG.xml',
	Text=>bmError.Text);
END_PROGRAM

(* POU zLibrary/ept/Programmbausteine/ST_CPU, ST *)
PROGRAM ST_CPU
VAR_INPUT
	iNumberOfFan			: INT := 1;
	iNumberOfCPU			: INT := 1;
	iLANIdx					: USINT;
END_VAR
VAR_IN_OUT

END_VAR
VAR_OUTPUT
	st_ctrl_out				: struct_ctrl_out;
	LNG					: enum_Lng:=DE;
END_VAR
VAR
	fb_ton_quitt				: TON;
	fb_state_entry			: ST_StateEntry;

	fbGetCPUUsage			: FB_MDP_CPU_Read;

	fbMDPNICRead			: FB_MDP_NIC_Read;	(* IP and MAC address *)

	fbGetRealTimeUsage	: TC_CpuUsage;

	fbGetHostName			:FB_GetHostName;

	nLastErrID	:UDINT;

	(* request cpu temperature *)
	fbGetCpuTemp			:FB_MDP_ReadElement;
	stMDP_Addr			:ST_MDP_Addr;		(* includes all address parameters without the Dynamic Module Id *)

	iCpu					:USINT;

	fbGetMainboardInfo		:FB_MDP_ReadElement;
	(* request fan speed *)
	fbGetFanSpeed			:FB_MDP_ReadElement;

	iFan					:USINT;

	fbGetTcInfo				:FB_MDP_TwinCAT_Read;

	b_temp								: BOOL;
	bm_CpuTemperatureToHigh 			: BOOL;
	bm_CpuUsageToHigh 				: BOOL;
	bm_FanSpeedToLow 				: BOOL;
	bm_RealTimeUsageToHigh 			: BOOL;
	bm_MainboardTemperatureToHigh 	: BOOL;

	(* visu *)
	s_Lng_Ip				: sData_Str:=(Description:='s_Lng_Ip');
	s_actual_IP_Adress		: sData_Str:=(Description:='s_actual_IP_Adress');
	b_DHCP				: sData_b:=(Description:='b_DHCP');
	s_Host_Name			: sData_Str:=(Description:='s_Host_Name');
	s_MAC_Address			: sData_Str:=(Description:='s_MAC_Address');
	s_Subnet_Mask			: sData_Str:=(Description:='s_Subnet_Mask');
	s_AMSNetId			: sData_Str:=(Description:='s_AMSNetId');
	i_Build					: sData_i16:=(Description:='i_Build', Unit:='no');
	i_RealTimeUsage		: sData_i16:=(Description:='i_RealTimeUsage', Unit:='%');
	i_FanSpeed				: ARRAY [0..4] OF sData_i16:=
										(Description:='i_FanSpeed[0]', Unit:='U/min'),
										(Description:='i_FanSpeed[1]', Unit:='U/min'),
										(Description:='i_FanSpeed[2]', Unit:='U/min'),
										(Description:='i_FanSpeed[3]', Unit:='U/min');
	i_CpuTemperature		: ARRAY [0..4] OF sData_i16:=
										(Description:='i_CpuTemperature[0]', Unit:='°C'),
										(Description:='i_CpuTemperature[1]', Unit:='°C'),
										(Description:='i_CpuTemperature[2]', Unit:='°C'),
										(Description:='i_CpuTemperature[3]', Unit:='°C');
	i_CpuUsage			: ARRAY [0..4] OF sData_i16:=
										(Description:='i_CpuUsage[0]', Unit:='%'),
										(Description:='i_CpuUsage[1]', Unit:='%'),
										(Description:='i_CpuUsage[2]', Unit:='%'),
										(Description:='i_CpuUsage[3]', Unit:='%');
	i_MainboardTemperature	: sData_i16:=(Description:='i_MainboardTemperature', Unit:='°C');


END_VAR
VAR_TEMP
	i				:INT;
END_VAR
(*======================================================
   ST: ST_CPU
 ------------------------------------------------------
   Auth: 	Thomas Vilgis    						 
   Date: 	24.05.2018    						     
   Rev.: 		1.0	
   Desc:		Der Baustein liest am Anfang den Hostnamen, die MAC-Adresse, IP-Adresse
			und die TwinCAT Infos aus. Danach werden in einem bestimmten Intervall
			die Echtzeitauslastung des TwinCATs, die CPU-Auslastung und die 
			CPU-Temperaturen ausgelesen. Außerdem die Drehzahl der Lüfter.

   Historie: 	
   Auth: 	Werner Friedl    						 
   Date: 	01.03.2021
		LNG auslesen aus der IP 
		16,17 und 18 => DE
		19 und 20 => CZ
		22 => EN
 ========================================================*)
(* Zeiten *)
fb_ton_quitt(IN:= , PT:= t#100ms, Q=> , ET=> );

(* Flanken *)

(* ======================================Schrittkette======================================== *)
fb_state_entry(	i16_pos:= 1);

CASE fb_state_entry.i16_step OF
(*=======================================================*)
	INIT_OBJ:
		IF	TD.ArtNo <> '' AND
			CURRENTLANGUAGE <> '' THEN
			IF	CURRENTLANGUAGE = 'DE' THEN
				s_Lng_Ip.str:='DE';
				LNG:=DE;
			ELSIF
				CURRENTLANGUAGE = 'EN' THEN
				s_Lng_Ip.str:='EN';
				LNG:=EN;
			ELSIF
				CURRENTLANGUAGE = 'CZ' THEN
				s_Lng_Ip.str:='CZ';
				LNG:=CZ;
			END_IF
			fb_state_entry.i16_next_step := INIT;
		END_IF

(*=======================================================*)
	INIT:
		IF fb_state_entry.E THEN
			fb_ton_quitt.IN := FALSE;
			st_ctrl_out.b_fehler := FALSE;
			st_ctrl_out.b_bereit := FALSE;
			st_ctrl_out.b_fertig := FALSE;
			st_ctrl_out.b_busy := FALSE;

			bm_CpuTemperatureToHigh := FALSE;
			bm_CpuUsageToHigh := FALSE;
			bm_FanSpeedToLow := FALSE;
			bm_RealTimeUsageToHigh := FALSE;
			bm_MainboardTemperatureToHigh := FALSE;

			fbGetCPUUsage.bExecute := FALSE;
			fbGetRealTimeUsage.START := FALSE;
			fbMDPNICRead.bExecute := FALSE;
			fbGetHostName.bExecute := FALSE;
			fbGetCpuTemp.bExecute := FALSE;
			fbGetFanSpeed.bExecute := FALSE;
			fbGetTcInfo.bExecute := FALSE;
			fbGetMainboardInfo.bExecute := FALSE;
			nLastErrID:=0;
			iLANIdx:=INT_TO_USINT(MP.ST00.LAN_no.i16);			(*0=LAN1, 1=LAN2, 2=LAN-USB*)
		END_IF

		(*-----------------------Weiterschaltbedingungen----------------------------*)
		IF 	fb_state_entry.fb_ton_Step.ET > t#10s THEN
			fb_state_entry.i16_next_step := 20;
		END_IF

(*=======================================================*)
	20:	fb_state_entry.s_debugtext:='Get Host Name ';

		IF fb_state_entry.E THEN
			fbGetHostName.bExecute := TRUE;
		END_IF

		(*-----------------------Weiterschaltbedingungen----------------------------*)
		IF fbGetHostName.bBusy THEN
			fbGetHostName.bExecute := FALSE;
			fb_state_entry.i16_next_step := 30;
		END_IF

(*=======================================================*)
	30:	fb_state_entry.s_debugtext:='Get Host Name  ';

		(*-----------------------Weiterschaltbedingungen----------------------------*)
		IF NOT fbGetHostName.bBusy THEN
			IF NOT fbGetHostName.bError THEN
				fb_state_entry.i16_next_step := 40;
			ELSE
				nLastErrID := fbGetHostName.nErrID;
				fb_state_entry.i16_next_step := FEHLER;
			END_IF
		END_IF

(*=======================================================*)
	40:	fb_state_entry.s_debugtext:='Get IP Adress und MAC-Adress';

		IF fb_state_entry.E THEN
			fbMDPNICRead.bExecute := TRUE;
		END_IF

		(*-----------------------Weiterschaltbedingungen----------------------------*)
		IF fbMDPNICRead.bBusy THEN
			fbMDPNICRead.bExecute := FALSE;
			fb_state_entry.i16_next_step := 50;
		END_IF

(*=======================================================*)
	50:	fb_state_entry.s_debugtext:='Get IP Adress und MAC-Adress ';

		(*-----------------------Weiterschaltbedingungen----------------------------*)
		IF 	NOT fbMDPNICRead.bBusy THEN
			IF NOT fbMDPNICRead.bError THEN
				fb_state_entry.i16_next_step := 60;
			ELSE
				nLastErrID := fbMDPNICRead.nErrID;
				fb_state_entry.i16_next_step := FEHLER;
			END_IF
		END_IF

(*=======================================================*)
	60:	fb_state_entry.s_debugtext:='Get IP Adress und MAC-Adress ';

		(*-----------------------Weiterschaltbedingungen----------------------------*)
		IF fb_state_entry.E THEN
			s_actual_IP_Adress.str := fbMDPNICRead.stMDP_ModuleContent.sIPAddress;
			s_MAC_Address.str := fbMDPNICRead.stMDP_ModuleContent.sMACAddress;
			s_Subnet_Mask.str := fbMDPNICRead.stMDP_ModuleContent.sSubnetMask;
			b_DHCP.b := fbMDPNICRead.stMDP_ModuleContent.bDHCP;
			s_Lng_Ip.str:=s_actual_IP_Adress.str;
			s_Lng_Ip.str:=RIGHT(	s_Lng_Ip.str,	LEN(s_Lng_Ip.str) - FIND(s_Lng_Ip.str,'.')	);
			s_Lng_Ip.str:=LEFT(s_Lng_Ip.str, 2);
			fb_state_entry.i16_next_step := 70;
			IF	s_Lng_Ip.str = '16' OR s_Lng_Ip.str = '17' OR s_Lng_Ip.str = '18' THEN	(*Peiting, Buching, Augsburg*)
				s_Lng_Ip.str:=CONCAT(s_Lng_Ip.str,' => DE');
				LNG:= DE;
				MP.ST00.LAN_no.i16:=USINT_TO_INT(iLANIdx);			(*0=LAN1, 1=LAN2, 2=LAN-USB*)
			ELSIF
				s_Lng_Ip.str = '22' THEN
				s_Lng_Ip.str:=CONCAT(s_Lng_Ip.str,' => EN');
				LNG:= EN;
				MP.ST00.LAN_no.i16:=USINT_TO_INT(iLANIdx);			(*0=LAN1, 1=LAN2, 2=LAN-USB*)
			ELSIF
				s_Lng_Ip.str = '19' OR s_Lng_Ip.str = '20' THEN
				s_Lng_Ip.str:=CONCAT(s_Lng_Ip.str,' => CZ');
				LNG:= CZ;
				MP.ST00.LAN_no.i16:=USINT_TO_INT(iLANIdx);			(*0=LAN1, 1=LAN2, 2=LAN-USB*)
			ELSE
				IF	iLANIdx<2 THEN
						iLANIdx:=iLANIdx + 1;
						fb_state_entry.i16_next_step := 40;
				END_IF
			END_IF
	END_IF

(*=======================================================*)
	70:	fb_state_entry.s_debugtext:='Get TwinCAT Info ';
		IF fb_state_entry.E THEN
			fbGetTcInfo.bExecute := TRUE;
		END_IF

		(*-----------------------Weiterschaltbedingungen----------------------------*)
		IF fbGetTcInfo.bBusy THEN
			fbGetTcInfo.bExecute := FALSE;
			fb_state_entry.i16_next_step := 80;
		END_IF

(*=======================================================*)
	80:	fb_state_entry.s_debugtext:='Get TwinCAT Info ';

		(*-----------------------Weiterschaltbedingungen----------------------------*)
		IF NOT fbGetTcInfo.bBusy THEN
			IF NOT fbGetTcInfo.bError THEN
				s_AMSNetId.str := fbGetTcInfo.stMDP_ModuleContent.sAmsNETid;
				i_Build.i16 := fbGetTcInfo.stMDP_ModuleContent.iBuild;
				fb_state_entry.i16_next_step := BEREIT;
			ELSE
				nLastErrID := fbGetTcInfo.nErrID;
				fb_state_entry.i16_next_step := FEHLER;
			END_IF
		END_IF

(*=======================================================*)
	BEREIT:	fb_state_entry.s_debugtext:='warte auf Start';

		IF fb_state_entry.E THEN
			st_ctrl_out.b_bereit := TRUE;
		END_IF

		(*-----------------------Weiterschaltbedingungen----------------------------*)
		IF 	iLANIdx <> INT_TO_USINT(MP.ST00.LAN_no.i16) THEN
			fb_state_entry.i16_next_step := INIT;
		END_IF

		IF 	fb_state_entry.fb_ton_Step.ET > t#10s THEN
			iCpu := 1;
			iFan := 1;
			fb_state_entry.i16_next_step := 110;
		END_IF

		IF fb_state_entry.X THEN
			st_ctrl_out.b_bereit := FALSE;
			st_ctrl_out.b_fertig := FALSE;
			st_ctrl_out.b_busy := TRUE;
		END_IF

(*=======================================================*)
	110:	fb_state_entry.s_debugtext:='Get Real Time Usage';

		IF fb_state_entry.E THEN
			fbGetRealTimeUsage.START := TRUE;
		END_IF

		(*-----------------------Weiterschaltbedingungen----------------------------*)
		IF 	fbGetRealTimeUsage.BUSY THEN
			fbGetRealTimeUsage.START := FALSE;
			fb_state_entry.i16_next_step := 120;
		END_IF

(*=======================================================*)
	120:	fb_state_entry.s_debugtext:='Get Real Time Usage';

		(*-----------------------Weiterschaltbedingungen----------------------------*)
		IF NOT fbGetRealTimeUsage.BUSY THEN
			IF NOT fbGetRealTimeUsage.ERR THEN
				i_RealTimeUsage.i16 := UDINT_TO_INT(fbGetRealTimeUsage.USAGE);
				fb_state_entry.i16_next_step := 130;
			ELSE
				nLastErrID := fbGetRealTimeUsage.ERRID;
				fb_state_entry.i16_next_step := FEHLER;
			END_IF
		END_IF

(*=======================================================*)
	130:	fb_state_entry.s_debugtext:='Get CPU Usage ';

		IF fb_state_entry.E THEN
			fbGetCPUUsage.bExecute := TRUE;
			fbGetCPUUsage.iModIdx := iCpu-1;		(* number of cpu *)
		END_IF

		(*-----------------------Weiterschaltbedingungen----------------------------*)
		IF fbGetCPUUsage.bBusy THEN
			fbGetCPUUsage.bExecute := FALSE;
			fb_state_entry.i16_next_step := 140;
		END_IF

(*=======================================================*)
	140:	fb_state_entry.s_debugtext:='Get CPU Usage';

		(*-----------------------Weiterschaltbedingungen----------------------------*)
		IF NOT fbGetCPUUsage.bBusy THEN
			IF NOT fbGetCPUUsage.bError THEN
				i_CpuUsage[iCpu-1].i16 := fbGetCPUUsage.stMDP_ModuleContent.iCPUusage;
				fb_state_entry.i16_next_step := 150;
			ELSE
				nLastErrID := fbGetCPUUsage.nErrId;
				fb_state_entry.i16_next_step := FEHLER;
			END_IF
		END_IF

(*=======================================================*)
	150:	fb_state_entry.s_debugtext:='Get CPU temperature';

		IF fb_state_entry.E THEN
			stMDP_Addr.nArea := INT_TO_BYTE(eMDP_Area_ConfigArea);
			stMDP_Addr.nTableId := 1;
			stMDP_Addr.nSubIdx := 3;			(* SubIndex 3 = cpu temperature *)
			fbGetCpuTemp.iModIdx := iCpu-1;		(* number of cpu *)
			fbGetCpuTemp.pDstBuf := ADR(i_CpuTemperature[iCpu-1].i16);
			fbGetCpuTemp.cbDstBufLen := SIZEOF(i_CpuTemperature[iCpu-1].i16);
			fbGetCpuTemp.bExecute := TRUE;
		END_IF

		(*-----------------------Weiterschaltbedingungen----------------------------*)
		IF fbGetCpuTemp.bBusy THEN
			fbGetCpuTemp.bExecute := FALSE;
			fb_state_entry.i16_next_step := 160;
		END_IF

(*=======================================================*)
	160:	fb_state_entry.s_debugtext:='Get CPU temperature';

		(*-----------------------Weiterschaltbedingungen----------------------------*)
		IF NOT fbGetCpuTemp.bBusy THEN
			IF NOT fbGetCpuTemp.bError THEN
				fb_state_entry.i16_next_step := 170;
			ELSE
				nLastErrID := fbGetCpuTemp.nErrId;
				fb_state_entry.i16_next_step := FEHLER;
			END_IF
		END_IF

(*=======================================================*)
	170:	fb_state_entry.s_debugtext:='warte';	(* Count CPU  *)
		IF fb_state_entry.E THEN
			iCpu := iCpu + 1;
		END_IF

		(*-----------------------Weiterschaltbedingungen----------------------------*)
		IF iCpu > iNumberOfCPU THEN
			fb_state_entry.i16_next_step := 180;
		ELSE
			fb_state_entry.i16_next_step := 130;
		END_IF

(*=======================================================*)
	180:	fb_state_entry.s_debugtext:='Get Fan speed ';

		IF fb_state_entry.E THEN
			stMDP_Addr.nArea := INT_TO_BYTE(eMDP_Area_ConfigArea);
			stMDP_Addr.nTableId := 1;
			stMDP_Addr.nSubIdx := 1;			(* SubIndex 1 = fan speed *)
			fbGetFanSpeed.iModIdx := iFan-1;		(* number of fan *)
			fbGetFanSpeed.pDstBuf := ADR(i_FanSpeed[iFan-1].i16);
			fbGetFanSpeed.cbDstBufLen := SIZEOF(i_FanSpeed[iFan-1].i16);
			fbGetFanSpeed.bExecute := TRUE;
		END_IF

		(*-----------------------Weiterschaltbedingungen----------------------------*)
		IF fbGetFanSpeed.bBusy THEN
			fbGetFanSpeed.bExecute := FALSE;
			fb_state_entry.i16_next_step := 190;
		END_IF

(*=======================================================*)
	190:	fb_state_entry.s_debugtext:='Get Fan speed';

		(*-----------------------Weiterschaltbedingungen----------------------------*)
		IF NOT fbGetFanSpeed.bBusy THEN
			IF NOT fbGetFanSpeed.bError THEN
				fb_state_entry.i16_next_step := 200;
			ELSE
				nLastErrID := fbGetFanSpeed.nErrId;
				fb_state_entry.i16_next_step := FEHLER;
			END_IF
		END_IF

(*=======================================================*)
	200:	fb_state_entry.s_debugtext:='Count Fan';

		IF fb_state_entry.E THEN
			iFan := iFan + 1;
		END_IF

		(*-----------------------Weiterschaltbedingungen----------------------------*)
		IF iFan > iNumberOfFan THEN
			fb_state_entry.i16_next_step := 210;
		ELSE
			fb_state_entry.i16_next_step := 180;
		END_IF

(*=======================================================*)
	210:	fb_state_entry.s_debugtext:='Get Mainboard Temperature';

		IF fb_state_entry.E THEN
			stMDP_Addr.nArea := INT_TO_BYTE(eMDP_Area_ConfigArea);
			stMDP_Addr.nTableId := 1;
			stMDP_Addr.nSubIdx := 10;			(* SubIndex 1 = mainboard temperature *)
			fbGetMainboardInfo.pDstBuf := ADR(i_MainboardTemperature.i16);
			fbGetMainboardInfo.cbDstBufLen := SIZEOF(i_MainboardTemperature.i16);
			fbGetMainboardInfo.bExecute := TRUE;
		END_IF

		(*-----------------------Weiterschaltbedingungen----------------------------*)
		IF fbGetMainboardInfo.bBusy THEN
			fbGetMainboardInfo.bExecute := FALSE;
			fb_state_entry.i16_next_step := 220;
		END_IF

(*=======================================================*)
	220:	fb_state_entry.s_debugtext:='GetMainboard Temperature ';

		(*-----------------------Weiterschaltbedingungen----------------------------*)
		IF NOT fbGetMainboardInfo.bBusy THEN
			IF NOT fbGetMainboardInfo.bError THEN
				fb_state_entry.i16_next_step := 230;
			ELSE
				nLastErrID := fbGetMainboardInfo.nErrId;
				fb_state_entry.i16_next_step := FEHLER;
			END_IF
		END_IF

(*=======================================================*)
	230:	fb_state_entry.s_debugtext:='evaluation';

		IF fb_state_entry.E THEN
			b_temp := FALSE;
			FOR i:=0 TO iNumberOfFan-1 DO
				IF i_FanSpeed[i].i16 < 5500 THEN
					b_temp := TRUE;
				END_IF
			END_FOR
			bm_FanSpeedToLow := b_temp;

			b_temp := FALSE;
			FOR i:=0 TO iNumberOfCPU-1 DO
				IF i_CpuTemperature[i].i16 > 80 THEN
					b_temp := TRUE;
				END_IF
			END_FOR
			bm_CpuTemperatureToHigh := b_temp;

			b_temp := FALSE;
			FOR i:=0 TO iNumberOfCPU-1 DO
				IF i_CpuUsage[i].i16 > 70 THEN
					b_temp := TRUE;
				END_IF
			END_FOR
			bm_CpuUsageToHigh := b_temp;

			bm_RealTimeUsageToHigh := i_RealTimeUsage.i16 > 30;

			bm_MainboardTemperatureToHigh := i_MainboardTemperature.i16 > 70;
		END_IF

		(*-----------------------Weiterschaltbedingungen----------------------------*)
		st_ctrl_out.b_fertig := TRUE;
		st_ctrl_out.b_busy := FALSE;
		fb_state_entry.i16_next_step := BEREIT;

(*=======================================================*)
	STOP, FEHLER:fb_state_entry.s_debugtext:=CONCAT('Error ID: ',UDINT_TO_STRING(nLastErrID));

		IF fb_state_entry.E THEN
			st_ctrl_out.b_fehler := fb_state_entry.i16_next_step = FEHLER;
			st_ctrl_out.b_gestoppt := fb_state_entry.i16_next_step = STOP;
			fb_ton_quitt.IN := FALSE;

		END_IF

		(*-----------------------Weiterschaltbedingungen----------------------------*)
		IF 	fb_state_entry.fb_ton_Step.ET > t#2s THEN
			st_ctrl_out.b_fehler := FALSE;
			st_ctrl_out.b_gestoppt := FALSE;
			fb_ton_quitt.IN := TRUE;
		END_IF
	
		IF 	fb_ton_quitt.Q THEN
			fb_ton_quitt.IN := FALSE;
			fb_state_entry.i16_next_step := INIT;
		END_IF

END_CASE

fb_state_entry(i16_pos:= 2 );

fbGetFanSpeed(
	bExecute:= ,
	stMDP_Addr:= stMDP_Addr,
	eModuleType:= eMDP_ModT_Fan,
	iModIdx:= ,
	tTimeout:= ,	(* default 5s *)
	sAmsNetId:= , (* wenn in AmsNetId nichts drin steht, wird immer die lokale genommen*)
	bBusy=> ,
	bError=> ,
	nErrID=> ,
	nCount=> ,
	stMDP_DynAddr=> ,
	iModuleTypeCount=> ,
	iModuleCount=> );

fbGetCpuTemp(
	bExecute:= ,
	stMDP_Addr:= stMDP_Addr,
	eModuleType:= eMDP_ModT_CPU,
	iModIdx:= ,
	pDstBuf     := ,
	cbDstBufLen := ,
	tTimeout:= ,	(* default 5s *)
	sAmsNetId:= , (* wenn in AmsNetId nichts drin steht, wird immer die lokale genommen*)
	bBusy=> ,
	bError=> , 
	nErrID=> ,
	nCount=> ,
	stMDP_DynAddr=> ,
	iModuleTypeCount=> ,
	iModuleCount=> );

fbGetCPUUsage(
	bExecute:= ,
	tTimeout:= ,	(* default 5s *)
	iModIdx:= ,
	sAmsNetId:= , (* wenn in AmsNetId nichts drin steht, wird immer die lokale genommen*)
	bBusy=> ,
	bError=> ,
	nErrID=> ,
	iErrPos=> ,
	stMDP_ModuleHeader=> ,
	stMDP_ModuleContent=> );

fbMDPNICRead(
	bExecute:= ,
	tTimeout:= , 	(* default 5s *)
	iModIdx:= iLANIdx, 	(*0=EtherCAT, 1=LAN muss aber nicht immer so sein*)
	sAmsNetId:= , (* wenn in AmsNetId nichts drin steht, wird immer die lokale genommen*)
	bBusy=> ,
	bError=> ,
	nErrID=> ,
	iErrPos=> ,
	stMDP_ModuleHeader=> ,
	stMDP_ModuleContent=> );

fbGetRealTimeUsage(
	NETID:= ,(* wenn in AmsNetId nichts drin steht, wird immer die lokale genommen*)
	START:= ,
	TMOUT:= ,	(* default 5s *)
	BUSY=> ,
	ERR=> ,
	ERRID=> ,
	USAGE=> );

fbGetHostName(
	sNetID:= ,(* wenn in AmsNetId nichts drin steht, wird immer die lokale genommen*)
	bExecute:= ,
	tTimeout:= , 	(* default 5s *)
	bBusy=> ,
	bError=> ,
	nErrID=> ,
	sHostName=> s_Host_Name.str);

fbGetTcInfo(
	bExecute:= , 
	tTimeout:= , 	(* default 5s *)
	iModIdx:= , 
	sAmsNetId:= , (* wenn in AmsNetId nichts drin steht, wird immer die lokale genommen*)
	bBusy=> ,
	bError=> , 
	nErrID=> ,
	iErrPos=> ,
	stMDP_ModuleHeader=> , 
	stMDP_ModuleContent=> );

fbGetMainboardInfo(
	bExecute:= ,
	stMDP_Addr:= stMDP_Addr,
	eModuleType:= eMDP_ModT_Mainboard,
	iModIdx:= ,
	pDstBuf:= ,
	cbDstBufLen:= ,
	tTimeout:= , 
	sAmsNetId:= ,(* wenn in AmsNetId nichts drin steht, wird immer die lokale genommen*)
	bBusy=> , 
	bError=> ,
	nErrID=> ,
	nCount=> , 
	stMDP_DynAddr=> , 
	iModuleTypeCount=> ,
	iModuleCount=> );

(*
IF	TD.ArtNo <> '' THEN
	(* Fehlermeldungen und Betriebsmeldungen ab dem Startindex in die globalen Meldungsarrays schreiben *)
	garr_stoermeldungen[st_config.i16_meld_startindex + 0] := FALSE;
	garr_stoermeldungen[st_config.i16_meld_startindex + 1] := FALSE;
	garr_stoermeldungen[st_config.i16_meld_startindex + 2] := FALSE;
	garr_stoermeldungen[st_config.i16_meld_startindex + 3] := FALSE;
	garr_stoermeldungen[st_config.i16_meld_startindex + 4] := FALSE;

	garr_betriebsmeldungen[st_config.i16_meld_startindex + 0] := bm_RealTimeUsageToHigh;
	garr_betriebsmeldungen[st_config.i16_meld_startindex + 1] := bm_CpuTemperatureToHigh;
	garr_betriebsmeldungen[st_config.i16_meld_startindex + 2] := bm_CpuUsageToHigh;
	garr_betriebsmeldungen[st_config.i16_meld_startindex + 3] := bm_FanSpeedToLow;
	garr_betriebsmeldungen[st_config.i16_meld_startindex + 4] := bm_MainboardTemperatureToHigh;

END_IF*)
END_PROGRAM

(* POU zLibrary/ept/ST_AutoCheckIn, ST *)
PROGRAM ST_AutoCheckIn
VAR_INPUT
	i_IntervalDay				: INT;		(*all  X Tagen, 0 = jeden Tag*)
END_VAR
VAR_OUTPUT
END_VAR
VAR
	fb_state_entry			: ST_StateEntry;
	NT_StartProcess 		: NT_StartProcess;
	s_uhrzeit				: STRING;
	s_tmpUhrzeit			: STRING;
	i_DayOfYear			: DINT;
	i_ErrId					: UDINT;
END_VAR
VAR_TEMP
	i						:INT:=1;
END_VAR
VAR CONSTANT
	NO_OF_AUTOCHECKIN	: INT :=5;

 	s_AutoCheckIn			:  ARRAY[1..NO_OF_AUTOCHECKIN] OF STRING:=
											'AutoCheckInDaten.bat',
											'AutoCheckInEpson.bat',
											'',
											'',
											''			;
END_VAR
(*======================================================
   FB: Start AutoCheckIn
 ------------------------------------------------------
   Auth: 		Werner Friedl   						 
   Date: 		10.11.2020  						     
   Rev.: 		1.0	
   Desc:		Mit diesem Programm können Komponenten im Versdog automatisch eingecheckt werden.
			Für den Check in benötigt man einen Bat- Datei. Diese liegt im Projektverzeichnis "Tools" und 
			muss für jede Komponente erstellt werden.
			Wenn mehrere Komponeten Eingecheckt werden sollen muss im Array "s_AutoCheckIn" die
			Bat Datei eingetragen werden.

			- die Input Variable "i_IntervalDay" legt den Seicherintervall in x Tagen fest.
			Wenn das Speichern nicht klappt, dann wird einen Tag später der nächste Versuch gemacht.

		Beispiel Aufruf:
		ST_AutoCheckIn( i_IntervalDay:=7 );

   Historie:   1.0

=======================================================*)

(* Uhrzei *)
s_uhrzeit:='';
s_uhrzeit:=CONCAT(s_uhrzeit, WORD_TO_STRING(gVarSystemtime.wHour));
s_uhrzeit:=CONCAT(s_uhrzeit, ':');
s_uhrzeit:=CONCAT(s_uhrzeit, WORD_TO_STRING(gVarSystemtime.wMinute));
s_uhrzeit:=CONCAT(s_uhrzeit, ':');
s_uhrzeit:=CONCAT(s_uhrzeit, WORD_TO_STRING(gVarSystemtime.wSecond));

(* Tag im Jahr *)
i_DayOfYear:=F_GetDOYOfYearMonthDay( gVarSystemtime.wYear, gVarSystemtime.wMonth, gVarSystemtime.wDay );

fb_state_entry(i16_pos:= 1);

CASE fb_state_entry.i16_step OF

(*=======================================================*)
INIT_OBJ:

	(*-----------------------Weiterschaltbedingungen----------------------------*)
	IF	i_DayOfYear <>0  AND
		fb_state_entry.fb_ton_Step.ET > t#5s THEN
		fb_state_entry.i16_next_step := 5;
	END_IF

(*=======================================================*)
5:
	(*-----------------------Weiterschaltbedingungen----------------------------*)
	IF	TD.ArtNo <>'' AND
		s_uhrzeit <> '00:00:00' AND s_uhrzeit <> ''  THEN
		IF	PersDaten.i_DayOfYearAutoCheckIn > i_DayOfYear THEN
			PersDaten.i_DayOfYearAutoCheckIn:= i_DayOfYear;
		END_IF
			fb_state_entry.i16_next_step := 6;
	END_IF

(*=======================================================*)
6:
	IF fb_state_entry.E THEN
		s_tmpUhrzeit:=s_uhrzeit;
		(*s_tmpUhrzeit:=REPLACE (s_tmpUhrzeit,'00',2,1);*)	(*nur in der Nacht sichern*)
	END_IF

	(*-----------------------Weiterschaltbedingungen----------------------------*)
	IF 	fb_state_entry.fb_ton_Step.ET > t#59s THEN
		IF	PersDaten.i_DayOfYearAutoCheckIn + i_IntervalDay < i_DayOfYear  THEN
			fb_state_entry.i16_next_step:=110;		(*gleich sicher, da das letzte Sichern zu lange her ist*)
		ELSE
			fb_state_entry.i16_next_step:=INIT;
		END_IF
	END_IF

(*=======================================================*)
INIT:
	IF 	fb_state_entry.E THEN
		;
	END_IF

	(*-----------------------Weiterschaltbedingungen----------------------------*)
	fb_state_entry.i16_next_step := BEREIT;

(*=======================================================*)
BEREIT: fb_state_entry.s_debugtext:='warte auf Start';

	IF 	fb_state_entry.E THEN
		;
	END_IF

	(*-----------------------Weiterschaltbedingungen----------------------------*)
	IF 	s_tmpUhrzeit=s_uhrzeit AND
		(PersDaten.i_DayOfYearAutoCheckIn + i_IntervalDay) <= i_DayOfYear THEN
		fb_state_entry.i16_next_step:=110;
	END_IF

	IF 	fb_state_entry.X THEN
		i:=0;
	END_IF

(*=======================================================*)
110:  fb_state_entry.s_debugtext:='Start Autocheckin';

	IF 	fb_state_entry.E THEN
		i:=i+1;
	END_IF

	IF	i = NO_OF_AUTOCHECKIN + 1 OR
		s_AutoCheckIn[i] = '' THEN
		fb_state_entry.i16_next_step:=200;
	ELSE
		fb_state_entry.i16_next_step:=120;
	END_IF

(*=======================================================*)
120:  fb_state_entry.s_debugtext:='Start Autocheckin';

	IF fb_state_entry.E THEN
		NT_StartProcess.START:=TRUE;
	END_IF

	(*-----------------------Weiterschaltbedingungen----------------------------*)
	IF 	NT_StartProcess.BUSY THEN
		fb_state_entry.i16_next_step:=130;
	END_IF

	IF 	fb_state_entry.X THEN
		NT_StartProcess.START:=FALSE;
	END_IF

(*=======================================================*)
130:  fb_state_entry.s_debugtext:='Warte auf fertig Autocheckin';

	IF 	NT_StartProcess.ERR THEN
		i_ErrId:=NT_StartProcess.ERRID;
		fb_state_entry.i16_next_step:=FEHLER;
	ELSIF
	 	fb_state_entry.fb_ton_Step.ET > t#5s AND
		NOT NT_StartProcess.BUSY AND
		NOT NT_StartProcess.ERR THEN
		fb_state_entry.i16_next_step:=110;
	END_IF

(*=======================================================*)
(*=======================================================*)
200:  fb_state_entry.s_debugtext:='Ende';

	(*-----------------------Weiterschaltbedingungen----------------------------*)
	PersDaten.i_DayOfYearAutoCheckIn:=i_DayOfYear;
	fb_state_entry.i16_next_step:=BEREIT;

(*=======================================================*)
STOP, FEHLER:
	IF 	fb_state_entry.E THEN
		IF	i_ErrId <> 0 THEN
		 	fb_state_entry.s_debugtext:=CONCAT('nErrId = ', UDINT_TO_STRING(i_ErrId)	);
		END_IF
		i_ErrId:=0;
	END_IF

	(*-----------------------Weiterschaltbedingungen----------------------------*)
	IF	fb_state_entry.fb_ton_Step.ET>t#1ms THEN
		fb_state_entry.i16_next_step := INIT;
	END_IF

END_CASE

fb_state_entry(i16_pos:= 2 );


(*Aufrufe======================================================*)
NT_StartProcess(
	NETID:='',
	PATHSTR		:='C:\Windows\System32\cmd.exe',
	DIRNAME		:=s_tools_path,
	COMNDLINE	:=CONCAT('/C start /b ', s_AutoCheckIn[i])	,
	START			:=,
	TMOUT			:=DEFAULT_ADS_TIMEOUT);
END_PROGRAM

(* POU zLibrary/ept/MainMenue/ST_MainMenue, ST *)
PROGRAM ST_MainMenue
VAR
	b_init					:BOOL:=FALSE;
	NT_StartProcess 		:NT_StartProcess;

	str_CurrentVisu_TD		:STRING:='TD_01_EDIT';

	FB_BtnTree				:FB_Btn;
END_VAR
IF NOT b_init THEN
	b_init:=TRUE;
END_IF

MainMenue_Btn_Init();
END_PROGRAM
ACTION MainMenue_Btn_Init:
(*=====================================================================*)
FB_BtnTree( Zoom:='MAIN',
			deaktivieren:=FALSE,
			unsichtbar:=FALSE,
			Btn=> Visu.MainMenue.BtnMainMenue);
(*=====================================================================*)
FB_BtnTree(Zoom:='MANUAL_MAIN',
			deaktivieren:=FALSE,
			unsichtbar:=FALSE,
			Btn=> Visu.MainMenue.BtnManual);
	(*=====================================================================*)
	FB_BtnTree(Zoom:='MANUAL_ST00_0',
				deaktivieren:=FALSE,
				unsichtbar:=FALSE,
				Btn=> Visu.MainMenue.BtnManual_ST00_0);
			(*=====================================================================*)
	FB_BtnTree(Zoom:='MANUAL_ST00_1',
				deaktivieren:=FALSE,
				unsichtbar:=	FALSE,
				Btn=> Visu.MainMenue.BtnManual_ST00_1);
	FB_BtnTree(Zoom:='MANUAL_ST00_2',
				deaktivieren:=FALSE,
				unsichtbar:=						gTypeCode<>312  AND gTypeCode <> 4991,
				Btn=> Visu.MainMenue.BtnManual_ST00_2);
	(*=====================================================================*)
	FB_BtnTree(Zoom:='MANUAL_ST02_0',
				deaktivieren:=FALSE,
				unsichtbar:=						gTypeCode<>312  AND gTypeCode <> 4991,
				Btn=> Visu.MainMenue.BtnManual_ST02_0);
	(*=====================================================================*)
	FB_BtnTree(Zoom:='MANUAL_ST03_0',
				deaktivieren:=FALSE,
				unsichtbar:=FALSE,
				Btn=> Visu.MainMenue.BtnManual_ST03_0);
		(*=====================================================================*)
		(*Visu Seiten abhängig vom Stecker zuweisen*)
		CASE  gTypeCode OF
			312,4991:	FB_BtnTree.Zoom:='MANUAL_ST03_2';		(*93pol, 102pol*)
			322:		FB_BtnTree.Zoom:='MANUAL_ST03_3';		(*160pol*)
			4871:	FB_BtnTree.Zoom:='MANUAL_ST03_4';		(*154pol*)
			4872:	FB_BtnTree.Zoom:='MANUAL_ST03_5';		(*154 Rasterplatte*)
			522:		FB_BtnTree.Zoom:='MANUAL_ST03_6';		(*206pol*)
			550:		FB_BtnTree.Zoom:='MANUAL_ST03_8';		(*92pol*)
			564:		FB_BtnTree.Zoom:='MANUAL_ST03_7';		(*124pol*)
			569:		FB_BtnTree.Zoom:='MANUAL_ST03_9';		(*46pol*)
			5632,5633:	FB_BtnTree.Zoom:='MANUAL_ST03_10';		(*NOX5 NOX6*)
			5631:	FB_BtnTree.Zoom:='MANUAL_ST03_11';		(*NOX4*)
			5731:	FB_BtnTree.Zoom:='MANUAL_ST03_12';		(*88pol*)
			575,5753,5754,5755:		FB_BtnTree.Zoom:='MANUAL_ST03_13';		(*7pol,9pol,6pol,9pol*)
			5732:	FB_BtnTree.Zoom:='MANUAL_ST03_14';		(*88pol AMG*)
			5771:	FB_BtnTree.Zoom:='MANUAL_ST03_15';		(*120pol*)
			5772:	FB_BtnTree.Zoom:='MANUAL_ST03_16';		(*21pol*)
			580:		FB_BtnTree.Zoom:='MANUAL_ST03_17';		(*191pol*)
			5831:	FB_BtnTree.Zoom:='MANUAL_ST03_19';		(*72pol*)
			5832:	FB_BtnTree.Zoom:='MANUAL_ST03_18';		(*48pol*)
			5841,4993:	FB_BtnTree.Zoom:='MANUAL_ST03_20';		(*268pol, 102pol neu*)
			5842:	FB_BtnTree.Zoom:='MANUAL_ST03_21';		(*268polRT*)
			598:	FB_BtnTree.Zoom:='MANUAL_ST03_22';		(*33pol*)

		ELSE
			FB_BtnTree.Zoom:='MANUAL_ST03_1';					(*74,91,168,35 pol*)
		END_CASE
		FB_BtnTree(
					deaktivieren:=FALSE,
					unsichtbar:=FALSE,
					Btn=> Visu.MainMenue.BtnManual_ST03_xx);
		(*=====================================================================*)
		(*Visu Seiten abhängig vom Stecker zuweisen (nur eintragen wenn eine zweite Seite benötigt wird)*)
		FB_BtnTree.unsichtbar:=	FALSE;
		CASE  gTypeCode OF
			322:		FB_BtnTree.Zoom:='MANUAL_ST03_3_2';	(*160pol*)
			569:		FB_BtnTree.Zoom:='MANUAL_ST03_9_2';	(*46pol*)
			575,5753,5754,5755:		FB_BtnTree.Zoom:='MANUAL_ST03_13_2';(*7pol,9pol,6pol,9pol*)
			5633:	FB_BtnTree.Zoom:='MANUAL_ST03_10_2';		(*NOX5 NOX6*)
(*			5841,4993:	FB_BtnTree.Zoom:='MANUAL_ST03_20_2';	*)	(*268pol, 102pol neu*)
			5842:	FB_BtnTree.Zoom:='MANUAL_ST03_21_2';	(*268polRT*)

		ELSE
			FB_BtnTree.unsichtbar:=	TRUE;
		END_CASE
		FB_BtnTree(
					deaktivieren:=FALSE,
					Btn=> Visu.MainMenue.BtnManual_ST03_xx_2);
	(*=====================================================================*)
	FB_BtnTree(	Zoom:='MANUAL_ST08_0',
				deaktivieren:=FALSE,
				unsichtbar:=FALSE,
				Btn=> Visu.MainMenue.BtnManual_ST08_0);
			(*=====================================================================*)
			FB_BtnTree(Zoom:='MANUAL_ST08_1',
						deaktivieren:=FALSE,
						unsichtbar:=FALSE,
						Btn=> Visu.MainMenue.BtnManual_ST08_1);
			(*=====================================================================*)
			FB_BtnTree(Zoom:='MANUAL_ST08_2',
						deaktivieren:=FALSE,
						unsichtbar:=FALSE,
						Btn=> Visu.MainMenue.BtnManual_ST08_2);
			(*=====================================================================*)
			FB_BtnTree(Zoom:='MANUAL_ST08_3',
						deaktivieren:=FALSE,
						unsichtbar:=FALSE,
						Btn=> Visu.MainMenue.BtnManual_ST08_3);
			(*=====================================================================*)
			FB_BtnTree(Zoom:='MANUAL_ST08_4',
						deaktivieren:=FALSE,
						unsichtbar:=FALSE,
						Btn=> Visu.MainMenue.BtnManual_ST08_4);
(*=====================================================================*)
FB_BtnTree(Zoom:='TD_MAIN',
			deaktivieren:=FALSE,
			unsichtbar:=FALSE,
			Btn=> Visu.MainMenue.BtnTD);
	(*=====================================================================*)
	FB_BtnTree(Zoom:='TD_01_EDIT',
				deaktivieren:=FALSE,
				unsichtbar:=FALSE,
				Btn=> Visu.MainMenue.BtnTD01_Edit);
	IF	FB_BtnTree.Zoom = CurrentVisu THEN
		str_CurrentVisu_TD:=FB_BtnTree.Zoom;
	 END_IF
	(*=====================================================================*)
	FB_BtnTree(Zoom:='TD_02_EDIT',
				deaktivieren:=FALSE,
				unsichtbar:=FALSE,
				Btn=> Visu.MainMenue.BtnTD02_Edit);
	IF	FB_BtnTree.Zoom = CurrentVisu THEN
		str_CurrentVisu_TD:=FB_BtnTree.Zoom;
	 END_IF
(*=====================================================================*)
FB_BtnTree(	Text:='MP_MAIN',
			Zoom:='MP_ST1',
			deaktivieren:=FALSE,
			unsichtbar:=FALSE,
			Btn=> Visu.MainMenue.BtnMP_Main);
	(*=====================================================================*)
	FB_BtnTree(Zoom:='MP_ST1',
			deaktivieren:=FALSE,
			unsichtbar:=FALSE,
			Btn=> Visu.MainMenue.BtnMP_ST1);
	(*=====================================================================*)
	FB_BtnTree(Zoom:='MP_ST2',
			deaktivieren:=FALSE,
			unsichtbar:=FALSE,
			Btn=> Visu.MainMenue.BtnMP_ST2);
	(*=====================================================================*)
	FB_BtnTree(Zoom:='MP_DATE',
				deaktivieren:=FALSE,
				unsichtbar:=FALSE,
				Btn=> Visu.MainMenue.BtnMP_Date);
	(*=====================================================================*)
	FB_BtnTree(Zoom:='MP_SERVICE',
				deaktivieren:=FALSE,
				unsichtbar:=FALSE,
				Btn=> Visu.MainMenue.BtnMP_Service);
(*=====================================================================*)
FB_BtnTree(Zoom:='SYSTEM_MAIN',
			deaktivieren:=FALSE,
			unsichtbar:=FALSE,
			Btn=> Visu.MainMenue.BtnSystem);
		(*=====================================================================*)
		FB_BtnTree(Zoom:='LOGFILE',
					deaktivieren:=FALSE,
					unsichtbar:=FALSE,
					Btn=> Visu.MainMenue.Btn_ErrorLog);
		(*Error Log wird mit vbs Skript gestartet*)
		NT_StartProcess(
			NETID:=,
			PATHSTR		:='C:\Windows\System32\wscript.exe',
			DIRNAME		:=s_tools_path,
			COMNDLINE	:='logfile.vbs',
			START			:=Visu.MainMenue.Btn_ErrorLog.tasten,
			TMOUT			:=T#10s);
		(*=====================================================================*)
		FB_BtnTree(Zoom:='SYSTEM_ERRORLIST',
					deaktivieren:=FALSE,
					unsichtbar:=FALSE,
					Btn=> Visu.MainMenue.Btn_ErrorList);
		(*=====================================================================*)
		FB_BtnTree(Zoom:='SYSTEM_GST',
					deaktivieren:=FALSE,
					unsichtbar:=FALSE,
					Btn=> Visu.MainMenue.Btn_Gst);
		(*=====================================================================*)
		FB_BtnTree(Zoom:='SYSTEM_STEP_DIAG',
			deaktivieren:=FALSE,
			unsichtbar:=FALSE,
			Btn=> Visu.MainMenue.Btn_Step_Diag);
		(*=====================================================================*)
		FB_BtnTree(Zoom:='SYSTEM_LNG',
					deaktivieren:=FALSE,
					unsichtbar:=FALSE,
					Btn=> Visu.MainMenue.Btn_Lng);
		(*=====================================================================*)
		FB_BtnTree(Zoom:='EXIT',
					deaktivieren:=FALSE,
					unsichtbar:=FALSE,
					Btn=> Visu.MainMenue.Btn_VisuBeenden);
END_ACTION

(* POU zLibrary/ept/MainMenue/FB_Btn, ST *)
FUNCTION_BLOCK FB_Btn
VAR_INPUT
	unsichtbar			: BOOL;
	deaktivieren		: BOOL;
	Zoom				: STRING(50);
	Text				: STRING(50);
END_VAR
VAR_OUTPUT
	Btn		:sButtonVisu_Tree;
END_VAR
VAR
END_VAR
IF 	Text = '' THEN
	Btn.Text:=Zoom;
ELSE
	Btn.Text:=Text;
END_IF
Text:='';
Btn.Zoom:=Zoom;
Btn.deaktivieren:=deaktivieren;
Btn.unsichtbar:=unsichtbar;

IF	Btn.Text = CurrentVisu THEN
	Btn.innenFarbe:=Color.darkgrey;
ELSE
	Btn.innenFarbe:=Color.lightgrey;
END_IF
IF	deaktivieren THEN
	Btn.Textfarbe:=Color.grey;
ELSE
	Btn.Textfarbe:=Color.black;
END_IF
END_FUNCTION_BLOCK

(* POU zLibrary/ept/ST_Path, ST *)
PROGRAM ST_Path
VAR_INPUT
	Start				: BOOL;
END_VAR
VAR_OUTPUT
	Done				: BOOL;
	Error_				: BOOL;
	nErrId				: UDINT;
END_VAR
VAR

	fb_state_entry		: ST_StateEntry;

	fb_xml_srv_read		: FB_XmlSrvReadByName;	(* XML Baustein zum Auslesen von Meldungen *)
	s_PLC_path_name		: T_MaxString;				(* Pfad füR XML Baustein *)

	len_str				: INT;
	mid_str				: STRING(1);

END_VAR
VAR_TEMP
	i					:INT;
END_VAR
(*======================================================
   FB: Start eines Win Prozess mit Prüfung 
 ------------------------------------------------------
   Auth: 		Werner Friedl   						 
   Date: 		06.03.2019   						     
   Rev.: 		1.0	
   Desc:		Mit diesem Programm wird der PLC Pfad und der Projektpfad sowie der PLC- Name eingelesen
		
		Achtung!
		unter 
			"Projekt => Optionen => TwinCAT "
			musse der Haken bei
			"Sympolbeschreibung als Datei herunterladen"
			gesetzt sein.

   Historie:   1.0

=======================================================*)
fb_state_entry(i16_pos:= 1);

CASE fb_state_entry.i16_step OF
(*=======================================================*)
INIT_OBJ:

	fb_state_entry.i16_next_step:=INIT;

(*=======================================================*)
INIT:  fb_state_entry.s_debugtext:='PLC Projektpfad mit Projektnamen aus TPY auslesen Achtung!! Bootprojekt muss erstellt sein';

	IF fb_state_entry.E THEN
		fb_xml_srv_read.sFilePath := 'C:\TwinCAT\Boot\CurrentPlc_1.tpy';
		fb_xml_srv_read.sXPath :='/PlcProjectInfo/ProjectInfo/Path';
		fb_xml_srv_read.sSymName := 'ST_Path.s_PLC_path_name';
		fb_xml_srv_read.bExecute := TRUE;
		Error_:=FALSE;
	END_IF

	(*-----------------------Weiterschaltbedingungen----------------------------*)
	IF fb_xml_srv_read.bBusy THEN
		fb_xml_srv_read.bExecute := FALSE;
		fb_state_entry.i16_next_step := 20;
	END_IF

(*=======================================================*)
20:  fb_state_entry.s_debugtext:='Lesevorgang erfolgreich?';

